SPLINE
SPL {X  -162.485, Y  +370.062, Z    +0.000, E1   +10.606, E3 +533690.258}
SPL {X  -162.818, Y  +379.636, Z    +0.000, E1    +5.115, E3 +533679.607}
SPL {X  -162.820, Y  +386.976, Z    +0.000, E1    +0.144, E3 +533678.706}
SPL {X  -162.820, Y  +391.982, Z    +0.000, E1    -3.443, E3 +533685.471}
SPL {X  -162.820, Y  +399.630, Z    +0.000, E1    -9.426, E3 +533687.978}
SPL {X  -162.820, Y  +408.127, Z    +0.000, E1   -18.417, E3 +533674.266}
SPL {X  -162.820, Y  +420.083, Z    +0.000, E1   -24.325, E3 +533694.742}
SPL {X  -162.820, Y  +428.527, Z    +0.000, E1   -26.988, E3 +533712.034}
SPL {X  -162.820, Y  +431.191, Z    +0.000, E1   -23.548, E3 +533746.887}
SPL {X  -162.820, Y  +432.946, Z    +0.000, E1   -22.795, E3 +533761.291}
SPL {X  -162.820, Y  +434.888, Z    +0.000, E1   -22.823, E3 +533770.697}
SPL {X  -162.820, Y  +436.834, Z    +0.000, E1   -22.779, E3 +533780.657}
SPL {X  -162.820, Y  +438.868, Z    +0.000, E1   -22.837, E3 +533790.311}
SPL {X  -162.820, Y  +441.351, Z    +0.000, E1   -22.805, E3 +533802.886}
SPL {X  -162.820, Y  +443.809, Z    +0.000, E1   -22.804, E3 +533815.052}
SPL {X  -162.820, Y  +446.105, Z    +0.000, E1   -22.815, E3 +533826.295}
SPL {X  -162.820, Y  +447.974, Z    +0.000, E1   -22.856, E3 +533835.198}
SPL {X  -162.820, Y  +449.911, Z    +0.000, E1   -22.774, E3 +533845.472}
SPL {X  -162.820, Y  +451.861, Z    +0.000, E1   -22.750, E3 +533855.320}
SPL {X  -162.820, Y  +454.167, Z    +0.000, E1   -22.842, E3 +533866.049}
SPL {X  -162.820, Y  +456.529, Z    +0.000, E1   -22.855, E3 +533877.578}
SPL {X  -162.820, Y  +458.725, Z    +0.000, E1   -22.793, E3 +533888.982}
SPL {X  -162.820, Y  +461.700, Z    +0.000, E1   -22.822, E3 +533903.605}
SPL {X  -162.820, Y  +464.633, Z    +0.000, E1   -22.813, E3 +533918.101}
SPL {X  -162.820, Y  +466.699, Z    +0.000, E1   -22.824, E3 +533928.147}
SPL {X  -162.820, Y  +468.655, Z    +0.000, E1   -22.858, E3 +533937.591}
SPL {X  -162.820, Y  +470.892, Z    +0.000, E1   -22.837, E3 +533948.830}
SPL {X  -162.820, Y  +472.726, Z    +0.000, E1   -22.777, E3 +533958.369}
SPL {X  -162.820, Y  +475.118, Z    +0.000, E1   -22.777, E3 +533970.340}
SPL {X  -162.820, Y  +478.177, Z    +0.000, E1   -22.834, E3 +533985.033}
SPL {X  -162.820, Y  +481.034, Z    +0.000, E1   -22.831, E3 +533999.170}
SPL {X  -162.820, Y  +483.391, Z    +0.000, E1   -22.793, E3 +534011.106}
SPL {X  -162.820, Y  +486.307, Z    +0.000, E1   -22.833, E3 +534025.360}
SPL {X  -162.820, Y  +488.828, Z    +0.000, E1   -22.793, E3 +534038.003}
SPL {X  -162.820, Y  +491.768, Z    +0.000, E1   -22.852, E3 +534052.300}
SPL {X  -162.820, Y  +495.526, Z    +0.000, E1   -22.833, E3 +534071.071}
SPL {X  -162.820, Y  +499.330, Z    +0.000, E1   -22.841, E3 +534089.852}
SPL {X  -162.820, Y  +503.049, Z    +0.000, E1   -22.823, E3 +534108.402}
SPL {X  -162.820, Y  +506.908, Z    +0.000, E1   -22.877, E3 +534127.072}
SPL {X  -162.820, Y  +510.068, Z    +0.000, E1   -22.761, E3 +534143.543}
SPL {X  -162.820, Y  +512.359, Z    +0.000, E1   -22.823, E3 +534154.275}
SPL {X  -162.820, Y  +513.873, Z    +0.000, E1   -22.800, E3 +534161.961}
SPL {X  -162.820, Y  +516.100, Z    +0.000, E1   -22.809, E3 +534173.038}
SPL {X  -162.820, Y  +518.662, Z    +0.000, E1   -22.847, E3 +534185.337}
SPL {X  -162.820, Y  +520.641, Z    +0.000, E1   -22.790, E3 +534195.578}
SPL {X  -162.820, Y  +523.535, Z    +0.000, E1   -22.857, E3 +534209.546}
SPL {X  -162.820, Y  +526.661, Z    +0.000, E1   -22.801, E3 +534225.371}
SPL {X  -162.820, Y  +528.725, Z    +0.000, E1   -22.770, E3 +534235.740}
SPL {X  -162.820, Y  +530.303, Z    +0.000, E1   -22.798, E3 +534243.359}
SPL {X  -162.820, Y  +532.614, Z    +0.000, E1   -22.828, E3 +534254.627}
SPL {X  -162.820, Y  +534.838, Z    +0.000, E1   -22.864, E3 +534265.256}
SPL {X  -162.820, Y  +536.882, Z    +0.000, E1   -22.782, E3 +534276.111}
SPL {X  -162.820, Y  +539.194, Z    +0.000, E1   -22.826, E3 +534287.160}
SPL {X  -162.820, Y  +541.555, Z    +0.000, E1   -22.817, E3 +534298.974}
SPL {X  -162.820, Y  +543.728, Z    +0.000, E1   -22.799, E3 +534309.832}
SPL {X  -162.820, Y  +545.925, Z    +0.000, E1   -22.803, E3 +534320.702}
SPL {X  -162.820, Y  +549.071, Z    +0.000, E1   -22.836, E3 +534336.229}
SPL {X  -162.820, Y  +553.089, Z    +0.000, E1   -22.838, E3 +534356.129}
SPL {X  -162.820, Y  +556.430, Z    +0.000, E1   -22.821, E3 +534372.630}
SPL {X  -162.820, Y  +558.974, Z    +0.000, E1   -22.806, E3 +534385.330}
SPL {X  -162.820, Y  +562.171, Z    +0.000, E1   -22.845, E3 +534401.028}
SPL {X  -162.820, Y  +565.170, Z    +0.000, E1   -22.801, E3 +534416.041}
SPL {X  -162.820, Y  +567.308, Z    +0.000, E1   -22.750, E3 +534427.057}
SPL {X  -162.820, Y  +570.378, Z    +0.000, E1   -22.843, E3 +534441.681}
SPL {X  -162.820, Y  +573.634, Z    +0.000, E1   -22.827, E3 +534457.825}
SPL {X  -162.820, Y  +576.228, Z    +0.000, E1   -22.814, E3 +534470.721}
SPL {X  -162.820, Y  +578.553, Z    +0.000, E1   -22.801, E3 +534482.337}
SPL {X  -162.820, Y  +581.064, Z    +0.000, E1   -22.823, E3 +534494.622}
SPL {X  -162.820, Y  +583.435, Z    +0.000, E1   -22.808, E3 +534506.443}
SPL {X  -162.820, Y  +585.410, Z    +0.000, E1   -22.764, E3 +534516.579}
SPL {X  -162.820, Y  +587.676, Z    +0.000, E1   -22.853, E3 +534527.094}
SPL {X  -162.820, Y  +590.707, Z    +0.000, E1   -22.855, E3 +534542.244}
SPL {X  -162.820, Y  +593.650, Z    +0.000, E1   -22.810, E3 +534557.004}
SPL {X  -162.820, Y  +595.830, Z    +0.000, E1   -22.828, E3 +534567.620}
SPL {X  -162.820, Y  +598.094, Z    +0.000, E1   -22.843, E3 +534578.733}
SPL {X  -162.820, Y  +600.420, Z    +0.000, E1   -22.826, E3 +534590.365}
SPL {X  -162.820, Y  +602.573, Z    +0.000, E1   -22.830, E3 +534600.950}
SPL {X  -162.820, Y  +604.828, Z    +0.000, E1   -22.784, E3 +534612.588}
SPL {X  -162.820, Y  +608.133, Z    +0.000, E1   -22.831, E3 +534628.706}
SPL {X  -162.820, Y  +611.103, Z    +0.000, E1   -22.785, E3 +534643.632}
SPL {X  -162.820, Y  +613.294, Z    +0.000, E1   -22.780, E3 +534654.505}
SPL {X  -162.820, Y  +615.356, Z    +0.000, E1   -22.799, E3 +534664.562}
SPL {X  -162.820, Y  +617.439, Z    +0.000, E1   -22.808, E3 +534674.820}
SPL {X  -162.820, Y  +619.665, Z    +0.000, E1   -22.817, E3 +534685.788}
SPL {X  -162.820, Y  +621.733, Z    +0.000, E1   -22.759, E3 +534696.512}
SPL {X  -162.820, Y  +624.076, Z    +0.000, E1   -22.774, E3 +534708.017}
SPL {X  -162.820, Y  +627.244, Z    +0.000, E1   -22.803, E3 +534723.700}
SPL {X  -162.820, Y  +630.349, Z    +0.000, E1   -22.766, E3 +534739.232}
SPL {X  -162.820, Y  +632.572, Z    +0.000, E1   -22.785, E3 +534750.038}
SPL {X  -162.820, Y  +634.507, Z    +0.000, E1   -22.784, E3 +534759.677}
SPL {X  -162.820, Y  +636.863, Z    +0.000, E1   -22.760, E3 +534771.599}
SPL {X  -162.820, Y  +640.111, Z    +0.000, E1   -22.809, E3 +534787.482}
SPL {X  -162.820, Y  +643.449, Z    +0.000, E1   -22.796, E3 +534804.000}
SPL {X  -162.820, Y  +645.630, Z    +0.000, E1   -22.795, E3 +534814.696}
SPL {X  -162.820, Y  +647.561, Z    +0.000, E1   -22.705, E3 +534825.147}
SPL {X  -162.820, Y  +651.051, Z    +0.000, E1   -22.833, E3 +534841.566}
SPL {X  -162.820, Y  +653.898, Z    +0.000, E1   -22.796, E3 +534855.752}
SPL {X  -162.820, Y  +656.161, Z    +0.000, E1   -22.812, E3 +534866.873}
SPL {X  -162.820, Y  +658.384, Z    +0.000, E1   -22.822, E3 +534877.740}
SPL {X  -162.820, Y  +660.215, Z    +0.000, E1   -22.649, E3 +534888.330}
SPL {X  -162.820, Y  +662.823, Z    +0.000, E1   -22.799, E3 +534900.038}
SPL {X  -162.820, Y  +665.862, Z    +0.000, E1   -22.864, E3 +534914.738}
SPL {X  -162.820, Y  +668.960, Z    +0.000, E1   -22.773, E3 +534930.688}
SPL {X  -162.820, Y  +672.333, Z    +0.000, E1   -22.837, E3 +534947.024}
SPL {X  -162.812, Y  +675.071, Z    +0.000, E1   -22.742, E3 +534961.170}
SPL {X  -162.773, Y  +677.428, Z    +0.000, E1   -22.762, E3 +534972.767}
SPL {X  -162.691, Y  +679.987, Z    +0.000, E1   -22.794, E3 +534985.180}
SPL {X  -162.604, Y  +681.880, Z    +0.000, E1   -22.691, E3 +534995.341}
SPL {X  -162.458, Y  +684.346, Z    +0.000, E1   -22.764, E3 +535007.135}
SPL {X  -162.296, Y  +686.547, Z    +0.000, E1   -22.660, E3 +535018.752}
SPL {X  -162.090, Y  +688.902, Z    +0.000, E1   -22.700, E3 +535030.260}
SPL {X  -161.474, Y  +694.390, Z    +0.000, E1   -24.298, E3 +535043.615}
SPL {X  -158.730, Y  +709.763, Z    +0.000, E1   -31.225, E3 +535054.954}
ENDSPLINE

SPLINE
SPL {X  -160.932, Y  +698.225, Z    +0.000, E1   -21.712, E3 +535086.063}
SPL {X  -161.917, Y  +690.622, Z    +0.000, E1   -16.445, E3 +535099.663}
ENDSPLINE

SPLINE
SPL {X  -161.349, Y  +695.340, Z    +0.000, E1   -18.625, E3 +535107.282}
ENDSPLINE

SPLINE
SPL {X  -162.534, Y  +683.153, Z    +0.000, E1   -10.475, E3 +535128.413}
SPL {X  -162.820, Y  +667.630, Z    +0.000, E1    -0.882, E3 +535122.389}
SPL {X  -162.820, Y  +661.883, Z    +0.000, E1    +3.373, E3 +535127.832}
SPL {X  -162.820, Y  +653.808, Z    +0.000, E1    +9.891, E3 +535125.524}
SPL {X  -162.820, Y  +632.548, Z    +0.000, E1   +27.446, E3 +535122.060}
ENDSPLINE

SPLINE
SPL {X  -162.820, Y  +638.080, Z    +0.000, E1   +18.858, E3 +535149.809}
ENDSPLINE

SPLINE
SPL {X  -162.820, Y  +623.278, Z    +0.000, E1   +28.723, E3 +535151.379}
SPL {X  -162.820, Y  +618.658, Z    +0.000, E1   +26.841, E3 +535179.988}
ENDSPLINE

SPLINE
SPL {X  -162.820, Y  +623.685, Z    +0.000, E1   +22.346, E3 +535192.295}
ENDSPLINE

SPLINE
SPL {X  -162.820, Y  +621.304, Z    +0.000, E1   +22.259, E3 +535205.110}
SPL {X  -162.820, Y  +618.758, Z    +0.000, E1   +22.239, E3 +535218.261}
SPL {X  -162.820, Y  +616.062, Z    +0.000, E1   +22.275, E3 +535231.681}
SPL {X  -162.820, Y  +613.536, Z    +0.000, E1   +22.242, E3 +535244.803}
SPL {X  -162.820, Y  +610.461, Z    +0.000, E1   +22.264, E3 +535260.434}
SPL {X  -162.820, Y  +607.796, Z    +0.000, E1   +22.261, E3 +535273.805}
SPL {X  -162.820, Y  +605.178, Z    +0.000, E1   +22.267, E3 +535287.289}
SPL {X  -162.820, Y  +602.350, Z    +0.000, E1   +22.224, E3 +535301.907}
SPL {X  -162.820, Y  +599.842, Z    +0.000, E1   +22.298, E3 +535314.058}
SPL {X  -162.820, Y  +597.194, Z    +0.000, E1   +22.253, E3 +535327.979}
SPL {X  -162.820, Y  +594.779, Z    +0.000, E1   +22.284, E3 +535339.883}
SPL {X  -162.820, Y  +592.389, Z    +0.000, E1   +22.245, E3 +535352.499}
SPL {X  -162.820, Y  +589.492, Z    +0.000, E1   +22.304, E3 +535366.684}
SPL {X  -162.820, Y  +587.447, Z    +0.000, E1   +22.279, E3 +535377.213}
SPL {X  -162.820, Y  +585.192, Z    +0.000, E1   +22.298, E3 +535388.623}
SPL {X  -162.820, Y  +582.610, Z    +0.000, E1   +22.234, E3 +535402.246}
SPL {X  -162.820, Y  +580.317, Z    +0.000, E1   +22.300, E3 +535413.300}
SPL {X  -162.820, Y  +578.878, Z    +0.000, E1   +22.272, E3 +535420.810}
SPL {X  -162.820, Y  +576.856, Z    +0.000, E1   +22.233, E3 +535431.568}
SPL {X  -162.820, Y  +574.811, Z    +0.000, E1   +22.236, E3 +535441.832}
SPL {X  -162.820, Y  +572.645, Z    +0.000, E1   +22.246, E3 +535452.927}
SPL {X  -162.820, Y  +570.282, Z    +0.000, E1   +22.231, E3 +535464.978}
SPL {X  -162.820, Y  +567.961, Z    +0.000, E1   +22.247, E3 +535476.767}
SPL {X  -162.820, Y  +564.506, Z    +0.000, E1   +22.298, E3 +535494.081}
SPL {X  -162.820, Y  +561.620, Z    +0.000, E1   +22.191, E3 +535509.462}
SPL {X  -162.820, Y  +559.515, Z    +0.000, E1   +22.273, E3 +535519.464}
SPL {X  -162.820, Y  +556.723, Z    +0.000, E1   +22.309, E3 +535533.548}
SPL {X  -162.820, Y  +554.378, Z    +0.000, E1   +22.288, E3 +535545.393}
SPL {X  -162.820, Y  +552.787, Z    +0.000, E1   +22.213, E3 +535554.215}
SPL {X  -162.820, Y  +550.871, Z    +0.000, E1   +22.229, E3 +535563.810}
SPL {X  -162.820, Y  +548.168, Z    +0.000, E1   +22.298, E3 +535577.146}
SPL {X  -162.820, Y  +545.860, Z    +0.000, E1   +22.216, E3 +535589.403}
SPL {X  -162.820, Y  +543.558, Z    +0.000, E1   +22.285, E3 +535600.634}
SPL {X  -162.820, Y  +541.633, Z    +0.000, E1   +22.257, E3 +535610.562}
SPL {X  -162.820, Y  +539.116, Z    +0.000, E1   +22.302, E3 +535623.172}
SPL {X  -162.820, Y  +535.523, Z    +0.000, E1   +22.266, E3 +535641.834}
SPL {X  -162.820, Y  +531.757, Z    +0.000, E1   +22.276, E3 +535660.889}
SPL {X  -162.820, Y  +527.980, Z    +0.000, E1   +22.326, E3 +535679.720}
SPL {X  -162.820, Y  +524.599, Z    +0.000, E1   +22.287, E3 +535697.117}
SPL {X  -162.820, Y  +522.011, Z    +0.000, E1   +22.282, E3 +535710.194}
SPL {X  -162.820, Y  +519.457, Z    +0.000, E1   +22.481, E3 +535721.483}
SPL {X  -162.820, Y  +506.285, Z    +0.000, E1   +28.538, E3 +535732.941}
SPL {X  -162.820, Y  +504.441, Z    +0.000, E1   +27.574, E3 +535747.284}
SPL {X  -162.820, Y  +502.813, Z    +0.000, E1   +26.013, E3 +535765.481}
SPL {X  -162.820, Y  +502.016, Z    +0.000, E1   +24.802, E3 +535777.824}
SPL {X  -162.820, Y  +501.060, Z    +0.000, E1   +24.081, E3 +535788.013}
SPL {X  -162.820, Y  +500.336, Z    +0.000, E1   +23.110, E3 +535799.153}
SPL {X  -162.820, Y  +499.240, Z    +0.000, E1   +22.316, E3 +535811.464}
SPL {X  -162.820, Y  +498.027, Z    +0.000, E1   +21.516, E3 +535824.372}
SPL {X  -162.820, Y  +495.897, Z    +0.000, E1   +21.662, E3 +535834.292}
SPL {X  -162.820, Y  +493.717, Z    +0.000, E1   +21.704, E3 +535845.398}
SPL {X  -162.820, Y  +491.396, Z    +0.000, E1   +21.707, E3 +535857.522}
SPL {X  -162.820, Y  +488.560, Z    +0.000, E1   +21.695, E3 +535872.632}
SPL {X  -162.820, Y  +485.661, Z    +0.000, E1   +21.712, E3 +535887.517}
SPL {X  -162.820, Y  +483.668, Z    +0.000, E1   +21.664, E3 +535898.344}
SPL {X  -162.820, Y  +481.739, Z    +0.000, E1   +21.704, E3 +535908.058}
SPL {X  -162.820, Y  +479.894, Z    +0.000, E1   +21.695, E3 +535917.845}
SPL {X  -162.820, Y  +477.685, Z    +0.000, E1   +21.656, E3 +535929.783}
SPL {X  -162.820, Y  +475.419, Z    +0.000, E1   +21.711, E3 +535941.136}
SPL {X  -162.820, Y  +473.301, Z    +0.000, E1   +21.712, E3 +535952.233}
SPL {X  -162.820, Y  +470.965, Z    +0.000, E1   +21.700, E3 +535964.578}
SPL {X  -162.820, Y  +469.036, Z    +0.000, E1   +21.695, E3 +535974.621}
SPL {X  -162.820, Y  +467.138, Z    +0.000, E1   +21.678, E3 +535984.793}
SPL {X  -162.820, Y  +465.011, Z    +0.000, E1   +21.692, E3 +535995.776}
SPL {X  -162.820, Y  +462.669, Z    +0.000, E1   +21.752, E3 +536007.556}
SPL {X  -162.820, Y  +460.725, Z    +0.000, E1   +21.689, E3 +536018.169}
SPL {X  -162.820, Y  +458.666, Z    +0.000, E1   +21.695, E3 +536028.981}
SPL {X  -162.820, Y  +456.431, Z    +0.000, E1   +21.708, E3 +536040.510}
SPL {X  -162.820, Y  +453.609, Z    +0.000, E1   +21.757, E3 +536055.044}
SPL {X  -162.820, Y  +450.610, Z    +0.000, E1   +21.698, E3 +536071.101}
SPL {X  -162.820, Y  +448.170, Z    +0.000, E1   +21.667, E3 +536084.122}
SPL {X  -162.820, Y  +446.246, Z    +0.000, E1   +21.696, E3 +536093.939}
SPL {X  -162.820, Y  +443.784, Z    +0.000, E1   +21.713, E3 +536106.726}
SPL {X  -162.820, Y  +440.567, Z    +0.000, E1   +21.731, E3 +536123.565}
SPL {X  -162.820, Y  +437.628, Z    +0.000, E1   +21.678, E3 +536139.229}
SPL {X  -162.820, Y  +434.473, Z    +0.000, E1   +21.747, E3 +536155.326}
SPL {X  -162.820, Y  +431.492, Z    +0.000, E1   +21.686, E3 +536171.274}
SPL {X  -162.820, Y  +429.074, Z    +0.000, E1   +21.710, E3 +536183.726}
SPL {X  -162.820, Y  +426.023, Z    +0.000, E1   +21.718, E3 +536199.794}
SPL {X  -162.820, Y  +422.986, Z    +0.000, E1   +21.685, E3 +536215.842}
SPL {X  -162.820, Y  +420.528, Z    +0.000, E1   +21.706, E3 +536228.492}
SPL {X  -162.820, Y  +418.116, Z    +0.000, E1   +21.761, E3 +536240.639}
SPL {X  -162.820, Y  +416.127, Z    +0.000, E1   +21.715, E3 +536251.344}
SPL {X  -162.820, Y  +414.361, Z    +0.000, E1   +21.613, E3 +536261.531}
SPL {X  -162.820, Y  +412.134, Z    +0.000, E1   +21.697, E3 +536272.476}
SPL {X  -162.820, Y  +409.248, Z    +0.000, E1   +21.741, E3 +536287.411}
SPL {X  -162.820, Y  +406.238, Z    +0.000, E1   +21.697, E3 +536303.379}
SPL {X  -162.820, Y  +404.001, Z    +0.000, E1   +21.723, E3 +536314.809}
SPL {X  -162.820, Y  +402.223, Z    +0.000, E1   +21.697, E3 +536324.294}
SPL {X  -162.820, Y  +400.348, Z    +0.000, E1   +21.713, E3 +536334.020}
SPL {X  -162.820, Y  +398.298, Z    +0.000, E1   +21.721, E3 +536344.635}
SPL {X  -162.820, Y  +396.371, Z    +0.000, E1   +21.713, E3 +536354.817}
SPL {X  -162.820, Y  +394.508, Z    +0.000, E1   +21.616, E3 +536365.373}
SPL {X  -162.820, Y  +392.435, Z    +0.000, E1   +21.681, E3 +536375.726}
SPL {X  -162.820, Y  +389.390, Z    +0.000, E1   +21.742, E3 +536391.333}
SPL {X  -162.820, Y  +386.818, Z    +0.000, E1   +21.679, E3 +536405.092}
SPL {X  -162.820, Y  +384.697, Z    +0.000, E1   +21.693, E3 +536416.162}
SPL {X  -162.820, Y  +382.288, Z    +0.000, E1   +21.742, E3 +536428.286}
SPL {X  -162.820, Y  +380.381, Z    +0.000, E1   +21.655, E3 +536439.010}
SPL {X  -162.808, Y  +378.512, Z    +0.000, E1   +21.736, E3 +536448.063}
SPL {X  -162.776, Y  +376.710, Z    +0.000, E1   +21.698, E3 +536457.862}
SPL {X  -162.707, Y  +374.438, Z    +0.000, E1   +21.688, E3 +536469.866}
SPL {X  -162.607, Y  +372.171, Z    +0.000, E1   +21.692, E3 +536481.666}
SPL {X  -162.494, Y  +370.197, Z    +0.000, E1   +21.655, E3 +536492.292}
SPL {X  -162.349, Y  +368.131, Z    +0.000, E1   +21.624, E3 +536503.410}
SPL {X  -162.161, Y  +365.866, Z    +0.000, E1   +21.642, E3 +536515.095}
SPL {X  -161.927, Y  +363.466, Z    +0.000, E1   +21.730, E3 +536526.867}
SPL {X  -160.290, Y  +351.907, Z    +0.000, E1   +27.562, E3 +536534.444}
SPL {X  -159.725, Y  +348.905, Z    +0.000, E1   +26.136, E3 +536559.679}
ENDSPLINE

SPLINE
SPL {X  -160.871, Y  +355.385, Z    +0.000, E1   +21.841, E3 +536568.522}
SPL {X  -161.833, Y  +362.603, Z    +0.000, E1   +17.021, E3 +536578.553}
ENDSPLINE

SPLINE
SPL {X  -160.786, Y  +354.842, Z    +0.000, E1   +19.274, E3 +536610.709}
ENDSPLINE

SPLINE
SPL {X  -162.485, Y  +370.062, Z    +0.000, E1   +10.606, E3 +536617.087}
SPL {X  -162.818, Y  +379.636, Z    +0.000, E1    +5.115, E3 +536606.436}
SPL {X  -162.820, Y  +386.976, Z    +0.000, E1    +0.144, E3 +536605.535}
SPL {X  -162.820, Y  +390.236, Z    +0.000, E1    -2.204, E3 +536611.594}
SPL {X  -162.820, Y  +393.415, Z    +0.000, E1    -4.587, E3 +536612.878}
SPL {X  -162.820, Y  +399.630, Z    +0.000, E1    -9.426, E3 +536614.807}
SPL {X  -162.820, Y  +408.127, Z    +0.000, E1   -18.417, E3 +536601.096}
SPL {X  -162.820, Y  +420.083, Z    +0.000, E1   -24.325, E3 +536621.571}
SPL {X  -162.820, Y  +428.527, Z    +0.000, E1   -26.988, E3 +536638.863}
SPL {X  -162.820, Y  +431.191, Z    +0.000, E1   -23.548, E3 +536673.716}
SPL {X  -162.820, Y  +432.946, Z    +0.000, E1   -22.795, E3 +536688.120}
SPL {X  -162.820, Y  +434.888, Z    +0.000, E1   -22.823, E3 +536697.527}
SPL {X  -162.820, Y  +436.834, Z    +0.000, E1   -22.779, E3 +536707.487}
SPL {X  -162.820, Y  +438.868, Z    +0.000, E1   -22.837, E3 +536717.140}
SPL {X  -162.820, Y  +441.351, Z    +0.000, E1   -22.805, E3 +536729.715}
SPL {X  -162.820, Y  +443.809, Z    +0.000, E1   -22.804, E3 +536741.882}
SPL {X  -162.820, Y  +446.105, Z    +0.000, E1   -22.815, E3 +536753.124}
SPL {X  -162.820, Y  +447.974, Z    +0.000, E1   -22.856, E3 +536762.027}
SPL {X  -162.820, Y  +449.911, Z    +0.000, E1   -22.774, E3 +536772.302}
SPL {X  -162.820, Y  +451.861, Z    +0.000, E1   -22.750, E3 +536782.149}
SPL {X  -162.820, Y  +454.167, Z    +0.000, E1   -22.842, E3 +536792.879}
SPL {X  -162.820, Y  +456.529, Z    +0.000, E1   -22.855, E3 +536804.407}
SPL {X  -162.820, Y  +458.725, Z    +0.000, E1   -22.793, E3 +536815.811}
SPL {X  -162.820, Y  +461.700, Z    +0.000, E1   -22.822, E3 +536830.434}
SPL {X  -162.820, Y  +464.633, Z    +0.000, E1   -22.813, E3 +536844.931}
SPL {X  -162.820, Y  +466.699, Z    +0.000, E1   -22.824, E3 +536854.977}
SPL {X  -162.820, Y  +468.655, Z    +0.000, E1   -22.858, E3 +536864.420}
SPL {X  -162.820, Y  +470.892, Z    +0.000, E1   -22.837, E3 +536875.659}
SPL {X  -162.820, Y  +473.485, Z    +0.000, E1   -22.806, E3 +536888.858}
SPL {X  -162.820, Y  +476.589, Z    +0.000, E1   -22.788, E3 +536904.379}
SPL {X  -162.820, Y  +478.914, Z    +0.000, E1   -22.821, E3 +536915.477}
SPL {X  -162.820, Y  +481.034, Z    +0.000, E1   -22.831, E3 +536926.000}
SPL {X  -162.820, Y  +484.256, Z    +0.000, E1   -22.840, E3 +536942.018}
SPL {X  -162.820, Y  +487.952, Z    +0.000, E1   -22.824, E3 +536960.448}
SPL {X  -162.820, Y  +491.768, Z    +0.000, E1   -22.852, E3 +536979.129}
SPL {X  -162.820, Y  +495.526, Z    +0.000, E1   -22.833, E3 +536997.900}
SPL {X  -162.820, Y  +499.330, Z    +0.000, E1   -22.841, E3 +537016.682}
SPL {X  -162.820, Y  +503.049, Z    +0.000, E1   -22.823, E3 +537035.231}
SPL {X  -162.820, Y  +506.908, Z    +0.000, E1   -22.877, E3 +537053.901}
SPL {X  -162.820, Y  +510.068, Z    +0.000, E1   -22.761, E3 +537070.373}
SPL {X  -162.820, Y  +512.359, Z    +0.000, E1   -22.823, E3 +537081.104}
SPL {X  -162.820, Y  +513.873, Z    +0.000, E1   -22.800, E3 +537088.791}
SPL {X  -162.820, Y  +516.100, Z    +0.000, E1   -22.809, E3 +537099.867}
SPL {X  -162.820, Y  +518.662, Z    +0.000, E1   -22.847, E3 +537112.166}
SPL {X  -162.820, Y  +520.641, Z    +0.000, E1   -22.790, E3 +537122.407}
SPL {X  -162.820, Y  +523.535, Z    +0.000, E1   -22.857, E3 +537136.376}
SPL {X  -162.820, Y  +526.661, Z    +0.000, E1   -22.801, E3 +537152.200}
SPL {X  -162.820, Y  +528.725, Z    +0.000, E1   -22.770, E3 +537162.569}
SPL {X  -162.820, Y  +530.303, Z    +0.000, E1   -22.798, E3 +537170.188}
SPL {X  -162.820, Y  +532.614, Z    +0.000, E1   -22.828, E3 +537181.457}
SPL {X  -162.820, Y  +534.838, Z    +0.000, E1   -22.864, E3 +537192.086}
SPL {X  -162.820, Y  +536.882, Z    +0.000, E1   -22.782, E3 +537202.941}
SPL {X  -162.820, Y  +539.194, Z    +0.000, E1   -22.826, E3 +537213.989}
SPL {X  -162.820, Y  +541.555, Z    +0.000, E1   -22.817, E3 +537225.803}
SPL {X  -162.820, Y  +543.728, Z    +0.000, E1   -22.799, E3 +537236.661}
SPL {X  -162.820, Y  +545.925, Z    +0.000, E1   -22.803, E3 +537247.531}
SPL {X  -162.820, Y  +548.328, Z    +0.000, E1   -22.796, E3 +537259.526}
SPL {X  -162.820, Y  +551.027, Z    +0.000, E1   -22.819, E3 +537272.719}
SPL {X  -162.820, Y  +553.721, Z    +0.000, E1   -22.807, E3 +537286.163}
SPL {X  -162.820, Y  +556.430, Z    +0.000, E1   -22.821, E3 +537299.459}
SPL {X  -162.820, Y  +559.675, Z    +0.000, E1   -22.837, E3 +537315.540}
SPL {X  -162.820, Y  +562.799, Z    +0.000, E1   -22.814, E3 +537331.046}
SPL {X  -162.820, Y  +565.170, Z    +0.000, E1   -22.801, E3 +537342.871}
SPL {X  -162.820, Y  +568.020, Z    +0.000, E1   -22.787, E3 +537357.257}
SPL {X  -162.820, Y  +570.992, Z    +0.000, E1   -22.834, E3 +537371.477}
SPL {X  -162.820, Y  +572.901, Z    +0.000, E1   -22.775, E3 +537381.345}
SPL {X  -162.820, Y  +575.638, Z    +0.000, E1   -22.855, E3 +537394.454}
SPL {X  -162.820, Y  +578.553, Z    +0.000, E1   -22.801, E3 +537409.167}
SPL {X  -162.820, Y  +581.064, Z    +0.000, E1   -22.823, E3 +537421.451}
SPL {X  -162.820, Y  +583.435, Z    +0.000, E1   -22.808, E3 +537433.273}
SPL {X  -162.820, Y  +585.410, Z    +0.000, E1   -22.764, E3 +537443.409}
SPL {X  -162.820, Y  +587.676, Z    +0.000, E1   -22.853, E3 +537453.923}
SPL {X  -162.820, Y  +589.682, Z    +0.000, E1   -22.776, E3 +537464.453}
SPL {X  -162.820, Y  +591.720, Z    +0.000, E1   -22.868, E3 +537473.764}
SPL {X  -162.820, Y  +593.650, Z    +0.000, E1   -22.810, E3 +537483.834}
SPL {X  -162.820, Y  +595.830, Z    +0.000, E1   -22.828, E3 +537494.449}
SPL {X  -162.820, Y  +598.094, Z    +0.000, E1   -22.843, E3 +537505.563}
SPL {X  -162.820, Y  +600.420, Z    +0.000, E1   -22.826, E3 +537517.194}
SPL {X  -162.820, Y  +602.573, Z    +0.000, E1   -22.830, E3 +537527.779}
SPL {X  -162.820, Y  +604.828, Z    +0.000, E1   -22.784, E3 +537539.417}
SPL {X  -162.820, Y  +607.142, Z    +0.000, E1   -22.808, E3 +537550.598}
SPL {X  -162.820, Y  +608.890, Z    +0.000, E1   -22.790, E3 +537559.423}
SPL {X  -162.820, Y  +611.103, Z    +0.000, E1   -22.785, E3 +537570.461}
SPL {X  -162.820, Y  +613.294, Z    +0.000, E1   -22.780, E3 +537581.334}
SPL {X  -162.820, Y  +615.356, Z    +0.000, E1   -22.799, E3 +537591.391}
SPL {X  -162.820, Y  +617.439, Z    +0.000, E1   -22.808, E3 +537601.649}
SPL {X  -162.820, Y  +619.665, Z    +0.000, E1   -22.817, E3 +537612.617}
SPL {X  -162.820, Y  +621.733, Z    +0.000, E1   -22.759, E3 +537623.342}
SPL {X  -162.820, Y  +624.076, Z    +0.000, E1   -22.774, E3 +537634.847}
SPL {X  -162.820, Y  +626.527, Z    +0.000, E1   -22.768, E3 +537647.089}
SPL {X  -162.820, Y  +629.758, Z    +0.000, E1   -22.800, E3 +537663.018}
SPL {X  -162.820, Y  +632.572, Z    +0.000, E1   -22.785, E3 +537676.867}
SPL {X  -162.820, Y  +634.507, Z    +0.000, E1   -22.784, E3 +537686.506}
SPL {X  -162.820, Y  +636.863, Z    +0.000, E1   -22.760, E3 +537698.429}
SPL {X  -162.820, Y  +639.254, Z    +0.000, E1   -22.767, E3 +537710.212}
SPL {X  -162.820, Y  +641.888, Z    +0.000, E1   -22.790, E3 +537723.159}
SPL {X  -162.820, Y  +644.915, Z    +0.000, E1   -22.818, E3 +537737.934}
SPL {X  -162.820, Y  +647.561, Z    +0.000, E1   -22.705, E3 +537751.976}
SPL {X  -162.820, Y  +649.758, Z    +0.000, E1   -22.780, E3 +537762.166}
SPL {X  -162.820, Y  +651.708, Z    +0.000, E1   -22.810, E3 +537771.660}
SPL {X  -162.820, Y  +653.898, Z    +0.000, E1   -22.796, E3 +537782.581}
SPL {X  -162.820, Y  +656.161, Z    +0.000, E1   -22.812, E3 +537793.703}
SPL {X  -162.820, Y  +658.384, Z    +0.000, E1   -22.822, E3 +537804.569}
SPL {X  -162.820, Y  +660.215, Z    +0.000, E1   -22.649, E3 +537815.159}
SPL {X  -162.820, Y  +662.823, Z    +0.000, E1   -22.799, E3 +537826.867}
SPL {X  -162.820, Y  +665.862, Z    +0.000, E1   -22.864, E3 +537841.567}
SPL {X  -162.820, Y  +668.960, Z    +0.000, E1   -22.773, E3 +537857.518}
SPL {X  -162.820, Y  +672.333, Z    +0.000, E1   -22.837, E3 +537873.854}
SPL {X  -162.812, Y  +675.071, Z    +0.000, E1   -22.742, E3 +537887.999}
SPL {X  -162.773, Y  +677.428, Z    +0.000, E1   -22.762, E3 +537899.596}
SPL {X  -162.691, Y  +679.987, Z    +0.000, E1   -22.794, E3 +537912.010}
SPL {X  -162.604, Y  +681.880, Z    +0.000, E1   -22.691, E3 +537922.170}
SPL {X  -162.458, Y  +684.346, Z    +0.000, E1   -22.764, E3 +537933.964}
SPL {X  -162.296, Y  +686.547, Z    +0.000, E1   -22.660, E3 +537945.581}
SPL {X  -162.090, Y  +688.902, Z    +0.000, E1   -22.700, E3 +537957.089}
SPL {X  -161.474, Y  +694.390, Z    +0.000, E1   -24.298, E3 +537970.444}
SPL {X  -158.553, Y  +710.529, Z    +0.000, E1   -30.890, E3 +537987.006}
ENDSPLINE

SPLINE
SPL {X  -161.215, Y  +696.305, Z    +0.000, E1   -20.575, E3 +538013.587}
SPL {X  -161.691, Y  +692.643, Z    +0.000, E1   -17.369, E3 +538029.775}
SPL {X  -162.534, Y  +683.153, Z    +0.000, E1   -10.475, E3 +538055.242}
SPL {X  -162.820, Y  +667.630, Z    +0.000, E1    -0.882, E3 +538049.218}
SPL {X  -162.820, Y  +661.883, Z    +0.000, E1    +3.373, E3 +538054.662}
SPL {X  -162.820, Y  +653.808, Z    +0.000, E1    +9.891, E3 +538052.353}
SPL {X  -162.820, Y  +632.548, Z    +0.000, E1   +27.446, E3 +538048.890}
ENDSPLINE

SPLINE
SPL {X  -162.820, Y  +638.080, Z    +0.000, E1   +18.858, E3 +538076.638}
ENDSPLINE

SPLINE
SPL {X  -162.820, Y  +623.278, Z    +0.000, E1   +28.723, E3 +538078.209}
SPL {X  -162.820, Y  +618.658, Z    +0.000, E1   +26.841, E3 +538106.817}
ENDSPLINE

SPLINE
SPL {X  -162.820, Y  +623.685, Z    +0.000, E1   +22.346, E3 +538119.124}
ENDSPLINE

SPLINE
SPL {X  -162.820, Y  +621.304, Z    +0.000, E1   +22.259, E3 +538131.939}
SPL {X  -162.820, Y  +618.758, Z    +0.000, E1   +22.239, E3 +538145.090}
SPL {X  -162.820, Y  +616.062, Z    +0.000, E1   +22.275, E3 +538158.511}
SPL {X  -162.820, Y  +613.536, Z    +0.000, E1   +22.242, E3 +538171.632}
SPL {X  -162.820, Y  +611.128, Z    +0.000, E1   +22.252, E3 +538183.803}
SPL {X  -162.820, Y  +608.428, Z    +0.000, E1   +22.255, E3 +538197.586}
SPL {X  -162.820, Y  +605.984, Z    +0.000, E1   +22.221, E3 +538210.223}
SPL {X  -162.820, Y  +603.020, Z    +0.000, E1   +22.272, E3 +538225.122}
SPL {X  -162.820, Y  +599.168, Z    +0.000, E1   +22.310, E3 +538244.390}
SPL {X  -162.820, Y  +596.569, Z    +0.000, E1   +22.222, E3 +538258.112}
SPL {X  -162.820, Y  +594.115, Z    +0.000, E1   +22.273, E3 +538270.337}
SPL {X  -162.820, Y  +591.721, Z    +0.000, E1   +22.239, E3 +538282.652}
SPL {X  -162.820, Y  +589.492, Z    +0.000, E1   +22.304, E3 +538293.513}
SPL {X  -162.820, Y  +587.447, Z    +0.000, E1   +22.279, E3 +538304.042}
SPL {X  -162.820, Y  +585.192, Z    +0.000, E1   +22.298, E3 +538315.452}
SPL {X  -162.820, Y  +582.610, Z    +0.000, E1   +22.234, E3 +538329.076}
SPL {X  -162.820, Y  +580.317, Z    +0.000, E1   +22.300, E3 +538340.130}
SPL {X  -162.820, Y  +578.878, Z    +0.000, E1   +22.272, E3 +538347.639}
SPL {X  -162.820, Y  +576.856, Z    +0.000, E1   +22.233, E3 +538358.397}
SPL {X  -162.820, Y  +573.830, Z    +0.000, E1   +22.272, E3 +538373.533}
SPL {X  -162.820, Y  +570.852, Z    +0.000, E1   +22.234, E3 +538388.993}
SPL {X  -162.820, Y  +568.608, Z    +0.000, E1   +22.253, E3 +538400.126}
SPL {X  -162.820, Y  +565.838, Z    +0.000, E1   +22.271, E3 +538414.357}
SPL {X  -162.820, Y  +562.162, Z    +0.000, E1   +22.252, E3 +538433.175}
SPL {X  -162.820, Y  +558.919, Z    +0.000, E1   +22.286, E3 +538449.338}
SPL {X  -162.820, Y  +555.548, Z    +0.000, E1   +22.322, E3 +538466.247}
SPL {X  -162.820, Y  +552.787, Z    +0.000, E1   +22.213, E3 +538481.044}
SPL {X  -162.820, Y  +550.136, Z    +0.000, E1   +22.258, E3 +538494.278}
SPL {X  -162.820, Y  +546.694, Z    +0.000, E1   +22.290, E3 +538511.600}
SPL {X  -162.820, Y  +543.558, Z    +0.000, E1   +22.285, E3 +538527.463}
SPL {X  -162.820, Y  +541.633, Z    +0.000, E1   +22.257, E3 +538537.391}
SPL {X  -162.820, Y  +539.116, Z    +0.000, E1   +22.302, E3 +538550.002}
SPL {X  -162.820, Y  +536.913, Z    +0.000, E1   +22.192, E3 +538561.926}
SPL {X  -162.820, Y  +534.880, Z    +0.000, E1   +22.252, E3 +538571.880}
SPL {X  -162.820, Y  +532.896, Z    +0.000, E1   +22.234, E3 +538582.040}
SPL {X  -162.820, Y  +531.056, Z    +0.000, E1   +22.251, E3 +538591.322}
SPL {X  -162.820, Y  +528.708, Z    +0.000, E1   +22.319, E3 +538602.704}
SPL {X  -162.820, Y  +525.932, Z    +0.000, E1   +22.258, E3 +538617.460}
SPL {X  -162.820, Y  +522.524, Z    +0.000, E1   +22.326, E3 +538634.184}
SPL {X  -162.820, Y  +519.457, Z    +0.000, E1   +22.481, E3 +538648.313}
SPL {X  -162.820, Y  +506.285, Z    +0.000, E1   +28.538, E3 +538659.771}
SPL {X  -162.820, Y  +504.441, Z    +0.000, E1   +27.574, E3 +538674.113}
SPL {X  -162.820, Y  +502.813, Z    +0.000, E1   +26.013, E3 +538692.310}
SPL {X  -162.820, Y  +502.016, Z    +0.000, E1   +24.802, E3 +538704.653}
SPL {X  -162.820, Y  +501.060, Z    +0.000, E1   +24.081, E3 +538714.843}
SPL {X  -162.820, Y  +499.934, Z    +0.000, E1   +22.814, E3 +538730.711}
SPL {X  -162.820, Y  +498.303, Z    +0.000, E1   +21.749, E3 +538747.967}
SPL {X  -162.820, Y  +495.897, Z    +0.000, E1   +21.662, E3 +538761.121}
SPL {X  -162.820, Y  +493.717, Z    +0.000, E1   +21.704, E3 +538772.227}
SPL {X  -162.820, Y  +491.396, Z    +0.000, E1   +21.707, E3 +538784.351}
SPL {X  -162.820, Y  +489.485, Z    +0.000, E1   +21.661, E3 +538794.699}
SPL {X  -162.820, Y  +487.723, Z    +0.000, E1   +21.665, E3 +538803.903}
SPL {X  -162.820, Y  +485.661, Z    +0.000, E1   +21.712, E3 +538814.346}
SPL {X  -162.820, Y  +482.775, Z    +0.000, E1   +21.716, E3 +538829.598}
SPL {X  -162.820, Y  +479.894, Z    +0.000, E1   +21.695, E3 +538844.675}
SPL {X  -162.820, Y  +477.685, Z    +0.000, E1   +21.656, E3 +538856.612}
SPL {X  -162.820, Y  +475.419, Z    +0.000, E1   +21.711, E3 +538867.965}
SPL {X  -162.820, Y  +473.301, Z    +0.000, E1   +21.712, E3 +538879.062}
SPL {X  -162.820, Y  +470.965, Z    +0.000, E1   +21.700, E3 +538891.407}
SPL {X  -162.820, Y  +469.036, Z    +0.000, E1   +21.695, E3 +538901.451}
SPL {X  -162.820, Y  +467.138, Z    +0.000, E1   +21.678, E3 +538911.622}
SPL {X  -162.820, Y  +465.011, Z    +0.000, E1   +21.692, E3 +538922.605}
SPL {X  -162.820, Y  +462.669, Z    +0.000, E1   +21.752, E3 +538934.385}
SPL {X  -162.820, Y  +460.725, Z    +0.000, E1   +21.689, E3 +538944.998}
SPL {X  -162.820, Y  +458.666, Z    +0.000, E1   +21.695, E3 +538955.810}
SPL {X  -162.820, Y  +456.431, Z    +0.000, E1   +21.708, E3 +538967.339}
SPL {X  -162.820, Y  +454.628, Z    +0.000, E1   +21.674, E3 +538977.057}
SPL {X  -162.820, Y  +452.690, Z    +0.000, E1   +21.773, E3 +538986.331}
SPL {X  -162.820, Y  +450.610, Z    +0.000, E1   +21.698, E3 +538997.930}
SPL {X  -162.820, Y  +448.170, Z    +0.000, E1   +21.667, E3 +539010.951}
SPL {X  -162.820, Y  +445.508, Z    +0.000, E1   +21.732, E3 +539024.469}
SPL {X  -162.820, Y  +442.443, Z    +0.000, E1   +21.712, E3 +539040.590}
SPL {X  -162.820, Y  +439.933, Z    +0.000, E1   +21.690, E3 +539053.871}
SPL {X  -162.820, Y  +437.628, Z    +0.000, E1   +21.678, E3 +539066.059}
SPL {X  -162.820, Y  +434.473, Z    +0.000, E1   +21.747, E3 +539082.155}
SPL {X  -162.820, Y  +431.492, Z    +0.000, E1   +21.686, E3 +539098.104}
SPL {X  -162.820, Y  +429.074, Z    +0.000, E1   +21.710, E3 +539110.556}
SPL {X  -162.820, Y  +426.023, Z    +0.000, E1   +21.718, E3 +539126.623}
SPL {X  -162.820, Y  +422.986, Z    +0.000, E1   +21.685, E3 +539142.671}
SPL {X  -162.820, Y  +420.528, Z    +0.000, E1   +21.706, E3 +539155.321}
SPL {X  -162.820, Y  +418.116, Z    +0.000, E1   +21.761, E3 +539167.468}
SPL {X  -162.820, Y  +416.127, Z    +0.000, E1   +21.715, E3 +539178.173}
SPL {X  -162.820, Y  +414.361, Z    +0.000, E1   +21.613, E3 +539188.360}
SPL {X  -162.820, Y  +411.450, Z    +0.000, E1   +21.710, E3 +539202.934}
SPL {X  -162.820, Y  +408.590, Z    +0.000, E1   +21.735, E3 +539217.559}
SPL {X  -162.820, Y  +406.238, Z    +0.000, E1   +21.697, E3 +539230.208}
SPL {X  -162.820, Y  +403.166, Z    +0.000, E1   +21.746, E3 +539246.014}
SPL {X  -162.820, Y  +400.348, Z    +0.000, E1   +21.713, E3 +539260.849}
SPL {X  -162.820, Y  +398.298, Z    +0.000, E1   +21.721, E3 +539271.465}
SPL {X  -162.820, Y  +396.371, Z    +0.000, E1   +21.713, E3 +539281.647}
SPL {X  -162.820, Y  +394.508, Z    +0.000, E1   +21.616, E3 +539292.202}
SPL {X  -162.820, Y  +391.777, Z    +0.000, E1   +21.714, E3 +539305.861}
SPL {X  -162.820, Y  +388.822, Z    +0.000, E1   +21.717, E3 +539321.181}
SPL {X  -162.820, Y  +386.818, Z    +0.000, E1   +21.679, E3 +539331.921}
SPL {X  -162.820, Y  +384.697, Z    +0.000, E1   +21.693, E3 +539342.991}
SPL {X  -162.820, Y  +382.288, Z    +0.000, E1   +21.742, E3 +539355.115}
SPL {X  -162.817, Y  +379.520, Z    +0.000, E1   +21.723, E3 +539369.952}
SPL {X  -162.776, Y  +376.710, Z    +0.000, E1   +21.698, E3 +539384.691}
SPL {X  -162.707, Y  +374.438, Z    +0.000, E1   +21.688, E3 +539396.695}
SPL {X  -162.607, Y  +372.171, Z    +0.000, E1   +21.692, E3 +539408.495}
SPL {X  -162.494, Y  +370.197, Z    +0.000, E1   +21.655, E3 +539419.121}
SPL {X  -162.349, Y  +368.131, Z    +0.000, E1   +21.624, E3 +539430.239}
SPL {X  -162.161, Y  +365.866, Z    +0.000, E1   +21.642, E3 +539441.924}
SPL {X  -161.651, Y  +361.024, Z    +0.000, E1   +22.970, E3 +539455.348}
SPL {X  -160.281, Y  +351.857, Z    +0.000, E1   +24.243, E3 +539490.687}
ENDSPLINE

SPLINE
SPL {X  -161.833, Y  +362.603, Z    +0.000, E1   +17.021, E3 +539505.383}
ENDSPLINE

SPLINE
SPL {X  -160.786, Y  +354.842, Z    +0.000, E1   +19.274, E3 +539537.538}
ENDSPLINE

SPLINE
SPL {X  -162.485, Y  +370.062, Z    +0.000, E1   +10.606, E3 +539543.916}
SPL {X  -162.818, Y  +379.636, Z    +0.000, E1    +5.115, E3 +539533.265}
SPL {X  -162.820, Y  +386.976, Z    +0.000, E1    +0.144, E3 +539532.364}
SPL {X  -162.820, Y  +390.236, Z    +0.000, E1    -2.204, E3 +539538.423}
SPL {X  -162.820, Y  +393.415, Z    +0.000, E1    -4.587, E3 +539539.707}
SPL {X  -162.820, Y  +399.630, Z    +0.000, E1    -9.426, E3 +539541.637}
SPL {X  -162.820, Y  +408.127, Z    +0.000, E1   -18.417, E3 +539527.925}
SPL {X  -162.820, Y  +420.083, Z    +0.000, E1   -24.325, E3 +539548.400}
SPL {X  -162.820, Y  +428.527, Z    +0.000, E1   -26.988, E3 +539565.693}
SPL {X  -162.820, Y  +431.336, Z    +0.000, E1   -24.162, E3 +539595.903}
SPL {X  -162.820, Y  +432.048, Z    +0.000, E1   -22.832, E3 +539610.406}
SPL {X  -162.820, Y  +434.888, Z    +0.000, E1   -22.823, E3 +539624.356}
SPL {X  -162.820, Y  +436.834, Z    +0.000, E1   -22.779, E3 +539634.316}
SPL {X  -162.820, Y  +438.868, Z    +0.000, E1   -22.837, E3 +539643.969}
SPL {X  -162.820, Y  +441.351, Z    +0.000, E1   -22.805, E3 +539656.545}
SPL {X  -162.820, Y  +443.809, Z    +0.000, E1   -22.804, E3 +539668.711}
SPL {X  -162.820, Y  +446.105, Z    +0.000, E1   -22.815, E3 +539679.953}
SPL {X  -162.820, Y  +447.974, Z    +0.000, E1   -22.856, E3 +539688.856}
SPL {X  -162.820, Y  +449.911, Z    +0.000, E1   -22.774, E3 +539699.131}
SPL {X  -162.820, Y  +451.861, Z    +0.000, E1   -22.750, E3 +539708.978}
SPL {X  -162.820, Y  +454.167, Z    +0.000, E1   -22.842, E3 +539719.708}
SPL {X  -162.820, Y  +456.529, Z    +0.000, E1   -22.855, E3 +539731.236}
SPL {X  -162.820, Y  +458.725, Z    +0.000, E1   -22.793, E3 +539742.641}
SPL {X  -162.820, Y  +461.700, Z    +0.000, E1   -22.822, E3 +539757.263}
SPL {X  -162.820, Y  +464.633, Z    +0.000, E1   -22.813, E3 +539771.760}
SPL {X  -162.820, Y  +466.699, Z    +0.000, E1   -22.824, E3 +539781.806}
SPL {X  -162.820, Y  +468.655, Z    +0.000, E1   -22.858, E3 +539791.250}
SPL {X  -162.820, Y  +470.892, Z    +0.000, E1   -22.837, E3 +539802.488}
SPL {X  -162.820, Y  +473.485, Z    +0.000, E1   -22.806, E3 +539815.687}
SPL {X  -162.820, Y  +476.589, Z    +0.000, E1   -22.788, E3 +539831.209}
SPL {X  -162.820, Y  +478.914, Z    +0.000, E1   -22.821, E3 +539842.307}
SPL {X  -162.820, Y  +481.034, Z    +0.000, E1   -22.831, E3 +539852.829}
SPL {X  -162.820, Y  +484.256, Z    +0.000, E1   -22.840, E3 +539868.848}
SPL {X  -162.820, Y  +487.014, Z    +0.000, E1   -22.789, E3 +539882.715}
SPL {X  -162.820, Y  +489.750, Z    +0.000, E1   -22.832, E3 +539896.089}
SPL {X  -162.820, Y  +493.233, Z    +0.000, E1   -22.844, E3 +539913.226}
SPL {X  -162.820, Y  +496.150, Z    +0.000, E1   -22.796, E3 +539927.945}
SPL {X  -162.820, Y  +498.661, Z    +0.000, E1   -22.828, E3 +539940.126}
SPL {X  -162.820, Y  +501.761, Z    +0.000, E1   -22.820, E3 +539955.695}
SPL {X  -162.820, Y  +505.323, Z    +0.000, E1   -22.838, E3 +539973.142}
SPL {X  -162.820, Y  +507.875, Z    +0.000, E1   -22.849, E3 +539985.509}
SPL {X  -162.820, Y  +510.068, Z    +0.000, E1   -22.761, E3 +539997.202}
SPL {X  -162.820, Y  +512.359, Z    +0.000, E1   -22.823, E3 +540007.933}
SPL {X  -162.820, Y  +514.562, Z    +0.000, E1   -22.806, E3 +540019.120}
SPL {X  -162.820, Y  +517.952, Z    +0.000, E1   -22.864, E3 +540035.518}
SPL {X  -162.820, Y  +520.641, Z    +0.000, E1   -22.790, E3 +540049.236}
SPL {X  -162.820, Y  +522.740, Z    +0.000, E1   -22.811, E3 +540059.479}
SPL {X  -162.820, Y  +524.628, Z    +0.000, E1   -22.846, E3 +540068.474}
SPL {X  -162.820, Y  +526.661, Z    +0.000, E1   -22.801, E3 +540079.029}
SPL {X  -162.820, Y  +529.662, Z    +0.000, E1   -22.810, E3 +540093.880}
SPL {X  -162.820, Y  +532.614, Z    +0.000, E1   -22.828, E3 +540108.286}
SPL {X  -162.820, Y  +534.838, Z    +0.000, E1   -22.864, E3 +540118.915}
SPL {X  -162.820, Y  +536.882, Z    +0.000, E1   -22.782, E3 +540129.770}
SPL {X  -162.820, Y  +539.194, Z    +0.000, E1   -22.826, E3 +540140.818}
SPL {X  -162.820, Y  +541.555, Z    +0.000, E1   -22.817, E3 +540152.633}
SPL {X  -162.820, Y  +543.728, Z    +0.000, E1   -22.799, E3 +540163.490}
SPL {X  -162.820, Y  +545.925, Z    +0.000, E1   -22.803, E3 +540174.360}
SPL {X  -162.820, Y  +548.328, Z    +0.000, E1   -22.796, E3 +540186.356}
SPL {X  -162.820, Y  +551.027, Z    +0.000, E1   -22.819, E3 +540199.549}
SPL {X  -162.820, Y  +553.721, Z    +0.000, E1   -22.807, E3 +540212.993}
SPL {X  -162.820, Y  +556.430, Z    +0.000, E1   -22.821, E3 +540226.289}
SPL {X  -162.820, Y  +559.675, Z    +0.000, E1   -22.837, E3 +540242.369}
SPL {X  -162.820, Y  +562.799, Z    +0.000, E1   -22.814, E3 +540257.875}
SPL {X  -162.820, Y  +565.170, Z    +0.000, E1   -22.801, E3 +540269.700}
SPL {X  -162.820, Y  +568.020, Z    +0.000, E1   -22.787, E3 +540284.087}
SPL {X  -162.820, Y  +570.992, Z    +0.000, E1   -22.834, E3 +540298.306}
SPL {X  -162.820, Y  +572.901, Z    +0.000, E1   -22.775, E3 +540308.174}
SPL {X  -162.820, Y  +575.638, Z    +0.000, E1   -22.855, E3 +540321.284}
SPL {X  -162.820, Y  +578.553, Z    +0.000, E1   -22.801, E3 +540335.996}
SPL {X  -162.820, Y  +581.064, Z    +0.000, E1   -22.823, E3 +540348.280}
SPL {X  -162.820, Y  +583.435, Z    +0.000, E1   -22.808, E3 +540360.102}
SPL {X  -162.820, Y  +585.410, Z    +0.000, E1   -22.764, E3 +540370.238}
SPL {X  -162.820, Y  +587.676, Z    +0.000, E1   -22.853, E3 +540380.752}
SPL {X  -162.820, Y  +589.682, Z    +0.000, E1   -22.776, E3 +540391.282}
SPL {X  -162.820, Y  +591.720, Z    +0.000, E1   -22.868, E3 +540400.593}
SPL {X  -162.820, Y  +593.650, Z    +0.000, E1   -22.810, E3 +540410.663}
SPL {X  -162.820, Y  +595.830, Z    +0.000, E1   -22.828, E3 +540421.279}
SPL {X  -162.820, Y  +598.094, Z    +0.000, E1   -22.843, E3 +540432.392}
SPL {X  -162.820, Y  +600.420, Z    +0.000, E1   -22.826, E3 +540444.023}
SPL {X  -162.820, Y  +602.573, Z    +0.000, E1   -22.830, E3 +540454.608}
SPL {X  -162.820, Y  +604.828, Z    +0.000, E1   -22.784, E3 +540466.247}
SPL {X  -162.820, Y  +607.142, Z    +0.000, E1   -22.808, E3 +540477.428}
SPL {X  -162.820, Y  +608.890, Z    +0.000, E1   -22.790, E3 +540486.252}
SPL {X  -162.820, Y  +611.103, Z    +0.000, E1   -22.785, E3 +540497.290}
SPL {X  -162.820, Y  +613.294, Z    +0.000, E1   -22.780, E3 +540508.163}
SPL {X  -162.820, Y  +615.356, Z    +0.000, E1   -22.799, E3 +540518.221}
SPL {X  -162.820, Y  +617.439, Z    +0.000, E1   -22.808, E3 +540528.479}
SPL {X  -162.820, Y  +619.665, Z    +0.000, E1   -22.817, E3 +540539.447}
SPL {X  -162.820, Y  +621.733, Z    +0.000, E1   -22.759, E3 +540550.171}
SPL {X  -162.820, Y  +624.076, Z    +0.000, E1   -22.774, E3 +540561.676}
SPL {X  -162.820, Y  +627.244, Z    +0.000, E1   -22.803, E3 +540577.358}
SPL {X  -162.820, Y  +630.349, Z    +0.000, E1   -22.766, E3 +540592.890}
SPL {X  -162.820, Y  +632.572, Z    +0.000, E1   -22.785, E3 +540603.697}
SPL {X  -162.820, Y  +634.507, Z    +0.000, E1   -22.784, E3 +540613.336}
SPL {X  -162.820, Y  +636.863, Z    +0.000, E1   -22.760, E3 +540625.258}
SPL {X  -162.820, Y  +640.111, Z    +0.000, E1   -22.809, E3 +540641.141}
SPL {X  -162.820, Y  +643.449, Z    +0.000, E1   -22.796, E3 +540657.658}
SPL {X  -162.820, Y  +645.630, Z    +0.000, E1   -22.795, E3 +540668.354}
SPL {X  -162.820, Y  +647.561, Z    +0.000, E1   -22.705, E3 +540678.805}
SPL {X  -162.820, Y  +649.758, Z    +0.000, E1   -22.780, E3 +540688.995}
SPL {X  -162.820, Y  +651.708, Z    +0.000, E1   -22.810, E3 +540698.490}
SPL {X  -162.820, Y  +653.898, Z    +0.000, E1   -22.796, E3 +540709.410}
SPL {X  -162.820, Y  +656.161, Z    +0.000, E1   -22.812, E3 +540720.532}
SPL {X  -162.820, Y  +658.384, Z    +0.000, E1   -22.822, E3 +540731.398}
SPL {X  -162.820, Y  +660.215, Z    +0.000, E1   -22.649, E3 +540741.989}
SPL {X  -162.820, Y  +662.823, Z    +0.000, E1   -22.799, E3 +540753.697}
SPL {X  -162.820, Y  +665.862, Z    +0.000, E1   -22.864, E3 +540768.396}
SPL {X  -162.820, Y  +668.960, Z    +0.000, E1   -22.773, E3 +540784.347}
SPL {X  -162.820, Y  +671.605, Z    +0.000, E1   -22.777, E3 +540797.421}
SPL {X  -162.817, Y  +674.515, Z    +0.000, E1   -22.816, E3 +540811.618}
SPL {X  -162.773, Y  +677.428, Z    +0.000, E1   -22.762, E3 +540826.426}
SPL {X  -162.691, Y  +679.987, Z    +0.000, E1   -22.794, E3 +540838.839}
SPL {X  -162.604, Y  +681.880, Z    +0.000, E1   -22.691, E3 +540849.000}
SPL {X  -162.458, Y  +684.346, Z    +0.000, E1   -22.764, E3 +540860.793}
SPL {X  -162.296, Y  +686.547, Z    +0.000, E1   -22.660, E3 +540872.410}
SPL {X  -162.090, Y  +688.902, Z    +0.000, E1   -22.700, E3 +540883.918}
SPL {X  -161.474, Y  +694.390, Z    +0.000, E1   -24.298, E3 +540897.273}
SPL {X  -158.553, Y  +710.529, Z    +0.000, E1   -30.890, E3 +540913.835}
ENDSPLINE

SPLINE
SPL {X  -161.215, Y  +696.305, Z    +0.000, E1   -20.575, E3 +540940.416}
SPL {X  -161.691, Y  +692.643, Z    +0.000, E1   -17.369, E3 +540956.604}
SPL {X  -162.534, Y  +683.153, Z    +0.000, E1   -10.475, E3 +540982.071}
SPL {X  -162.820, Y  +667.630, Z    +0.000, E1    -0.882, E3 +540976.048}
SPL {X  -162.820, Y  +661.883, Z    +0.000, E1    +3.373, E3 +540981.491}
SPL {X  -162.820, Y  +653.808, Z    +0.000, E1    +9.891, E3 +540979.182}
SPL {X  -162.820, Y  +632.548, Z    +0.000, E1   +27.446, E3 +540975.719}
ENDSPLINE

SPLINE
SPL {X  -162.820, Y  +638.080, Z    +0.000, E1   +18.858, E3 +541003.467}
ENDSPLINE

SPLINE
SPL {X  -162.820, Y  +623.278, Z    +0.000, E1   +28.723, E3 +541005.038}
SPL {X  -162.820, Y  +618.658, Z    +0.000, E1   +26.841, E3 +541033.647}
ENDSPLINE

SPLINE
SPL {X  -162.820, Y  +623.685, Z    +0.000, E1   +22.346, E3 +541045.954}
ENDSPLINE

SPLINE
SPL {X  -162.820, Y  +621.304, Z    +0.000, E1   +22.259, E3 +541058.769}
SPL {X  -162.820, Y  +618.758, Z    +0.000, E1   +22.239, E3 +541071.919}
SPL {X  -162.820, Y  +616.062, Z    +0.000, E1   +22.275, E3 +541085.340}
SPL {X  -162.820, Y  +613.536, Z    +0.000, E1   +22.242, E3 +541098.462}
SPL {X  -162.820, Y  +610.461, Z    +0.000, E1   +22.264, E3 +541114.093}
SPL {X  -162.820, Y  +607.796, Z    +0.000, E1   +22.261, E3 +541127.464}
SPL {X  -162.820, Y  +605.178, Z    +0.000, E1   +22.267, E3 +541140.948}
SPL {X  -162.820, Y  +602.350, Z    +0.000, E1   +22.224, E3 +541155.565}
SPL {X  -162.820, Y  +599.842, Z    +0.000, E1   +22.298, E3 +541167.716}
SPL {X  -162.820, Y  +597.194, Z    +0.000, E1   +22.253, E3 +541181.637}
SPL {X  -162.820, Y  +594.779, Z    +0.000, E1   +22.284, E3 +541193.541}
SPL {X  -162.820, Y  +593.320, Z    +0.000, E1   +22.199, E3 +541201.645}
SPL {X  -162.820, Y  +591.031, Z    +0.000, E1   +22.283, E3 +541212.736}
SPL {X  -162.820, Y  +588.026, Z    +0.000, E1   +22.301, E3 +541227.863}
SPL {X  -162.820, Y  +585.899, Z    +0.000, E1   +22.286, E3 +541238.665}
SPL {X  -162.820, Y  +583.204, Z    +0.000, E1   +22.278, E3 +541252.688}
SPL {X  -162.820, Y  +579.691, Z    +0.000, E1   +22.312, E3 +541270.176}
SPL {X  -162.820, Y  +577.460, Z    +0.000, E1   +22.218, E3 +541282.163}
SPL {X  -162.820, Y  +575.394, Z    +0.000, E1   +22.240, E3 +541292.588}
SPL {X  -162.820, Y  +572.645, Z    +0.000, E1   +22.246, E3 +541306.586}
SPL {X  -162.820, Y  +570.282, Z    +0.000, E1   +22.231, E3 +541318.636}
SPL {X  -162.820, Y  +567.961, Z    +0.000, E1   +22.247, E3 +541330.426}
SPL {X  -162.820, Y  +564.506, Z    +0.000, E1   +22.298, E3 +541347.740}
SPL {X  -162.820, Y  +561.620, Z    +0.000, E1   +22.191, E3 +541363.121}
SPL {X  -162.820, Y  +558.919, Z    +0.000, E1   +22.286, E3 +541376.167}
SPL {X  -162.820, Y  +555.548, Z    +0.000, E1   +22.322, E3 +541393.076}
SPL {X  -162.820, Y  +552.787, Z    +0.000, E1   +22.213, E3 +541407.874}
SPL {X  -162.820, Y  +550.136, Z    +0.000, E1   +22.258, E3 +541421.107}
SPL {X  -162.820, Y  +546.694, Z    +0.000, E1   +22.290, E3 +541438.429}
SPL {X  -162.820, Y  +543.558, Z    +0.000, E1   +22.285, E3 +541454.292}
SPL {X  -162.820, Y  +541.633, Z    +0.000, E1   +22.257, E3 +541464.220}
SPL {X  -162.820, Y  +539.116, Z    +0.000, E1   +22.302, E3 +541476.831}
SPL {X  -162.820, Y  +536.913, Z    +0.000, E1   +22.192, E3 +541488.756}
SPL {X  -162.820, Y  +534.880, Z    +0.000, E1   +22.252, E3 +541498.709}
SPL {X  -162.820, Y  +532.896, Z    +0.000, E1   +22.234, E3 +541508.869}
SPL {X  -162.820, Y  +531.056, Z    +0.000, E1   +22.251, E3 +541518.151}
SPL {X  -162.820, Y  +528.708, Z    +0.000, E1   +22.319, E3 +541529.533}
SPL {X  -162.820, Y  +525.932, Z    +0.000, E1   +22.258, E3 +541544.289}
SPL {X  -162.820, Y  +522.524, Z    +0.000, E1   +22.326, E3 +541561.013}
SPL {X  -162.820, Y  +519.457, Z    +0.000, E1   +22.481, E3 +541575.142}
SPL {X  -162.820, Y  +506.285, Z    +0.000, E1   +28.538, E3 +541586.600}
SPL {X  -162.820, Y  +504.441, Z    +0.000, E1   +27.574, E3 +541600.942}
SPL {X  -162.820, Y  +503.215, Z    +0.000, E1   +26.369, E3 +541614.449}
SPL {X  -162.820, Y  +502.265, Z    +0.000, E1   +25.287, E3 +541626.931}
SPL {X  -162.820, Y  +501.060, Z    +0.000, E1   +24.081, E3 +541641.672}
SPL {X  -162.820, Y  +500.336, Z    +0.000, E1   +23.110, E3 +541652.812}
SPL {X  -162.820, Y  +499.240, Z    +0.000, E1   +22.316, E3 +541665.122}
SPL {X  -162.820, Y  +498.027, Z    +0.000, E1   +21.516, E3 +541678.030}
SPL {X  -162.820, Y  +495.897, Z    +0.000, E1   +21.662, E3 +541687.950}
SPL {X  -162.820, Y  +493.717, Z    +0.000, E1   +21.704, E3 +541699.057}
SPL {X  -162.820, Y  +491.396, Z    +0.000, E1   +21.707, E3 +541711.181}
SPL {X  -162.820, Y  +488.560, Z    +0.000, E1   +21.695, E3 +541726.290}
SPL {X  -162.820, Y  +485.661, Z    +0.000, E1   +21.712, E3 +541741.175}
SPL {X  -162.820, Y  +483.668, Z    +0.000, E1   +21.664, E3 +541752.003}
SPL {X  -162.820, Y  +481.739, Z    +0.000, E1   +21.704, E3 +541761.717}
SPL {X  -162.820, Y  +479.894, Z    +0.000, E1   +21.695, E3 +541771.504}
SPL {X  -162.820, Y  +477.685, Z    +0.000, E1   +21.656, E3 +541783.441}
SPL {X  -162.820, Y  +475.419, Z    +0.000, E1   +21.711, E3 +541794.794}
SPL {X  -162.820, Y  +473.301, Z    +0.000, E1   +21.712, E3 +541805.891}
SPL {X  -162.820, Y  +470.965, Z    +0.000, E1   +21.700, E3 +541818.236}
SPL {X  -162.820, Y  +469.036, Z    +0.000, E1   +21.695, E3 +541828.280}
SPL {X  -162.820, Y  +467.138, Z    +0.000, E1   +21.678, E3 +541838.452}
SPL {X  -162.820, Y  +465.011, Z    +0.000, E1   +21.692, E3 +541849.434}
SPL {X  -162.820, Y  +462.669, Z    +0.000, E1   +21.752, E3 +541861.215}
SPL {X  -162.820, Y  +460.725, Z    +0.000, E1   +21.689, E3 +541871.828}
SPL {X  -162.820, Y  +458.666, Z    +0.000, E1   +21.695, E3 +541882.640}
SPL {X  -162.820, Y  +456.431, Z    +0.000, E1   +21.708, E3 +541894.168}
SPL {X  -162.820, Y  +454.628, Z    +0.000, E1   +21.674, E3 +541903.886}
SPL {X  -162.820, Y  +452.690, Z    +0.000, E1   +21.773, E3 +541913.160}
SPL {X  -162.820, Y  +450.610, Z    +0.000, E1   +21.698, E3 +541924.759}
SPL {X  -162.820, Y  +448.170, Z    +0.000, E1   +21.667, E3 +541937.780}
SPL {X  -162.820, Y  +446.246, Z    +0.000, E1   +21.696, E3 +541947.598}
SPL {X  -162.820, Y  +443.784, Z    +0.000, E1   +21.713, E3 +541960.384}
SPL {X  -162.820, Y  +440.567, Z    +0.000, E1   +21.731, E3 +541977.224}
SPL {X  -162.820, Y  +437.628, Z    +0.000, E1   +21.678, E3 +541992.888}
SPL {X  -162.820, Y  +435.262, Z    +0.000, E1   +21.727, E3 +542004.824}
SPL {X  -162.820, Y  +433.510, Z    +0.000, E1   +21.692, E3 +542014.237}
SPL {X  -162.820, Y  +431.492, Z    +0.000, E1   +21.686, E3 +542024.933}
SPL {X  -162.820, Y  +429.074, Z    +0.000, E1   +21.710, E3 +542037.385}
SPL {X  -162.820, Y  +426.023, Z    +0.000, E1   +21.718, E3 +542053.453}
SPL {X  -162.820, Y  +422.986, Z    +0.000, E1   +21.685, E3 +542069.500}
SPL {X  -162.820, Y  +420.528, Z    +0.000, E1   +21.706, E3 +542082.150}
SPL {X  -162.820, Y  +418.116, Z    +0.000, E1   +21.761, E3 +542094.297}
SPL {X  -162.820, Y  +416.127, Z    +0.000, E1   +21.715, E3 +542105.003}
SPL {X  -162.820, Y  +414.361, Z    +0.000, E1   +21.613, E3 +542115.190}
SPL {X  -162.820, Y  +411.450, Z    +0.000, E1   +21.710, E3 +542129.763}
SPL {X  -162.820, Y  +408.590, Z    +0.000, E1   +21.735, E3 +542144.389}
SPL {X  -162.820, Y  +406.238, Z    +0.000, E1   +21.697, E3 +542157.038}
SPL {X  -162.820, Y  +403.166, Z    +0.000, E1   +21.746, E3 +542172.844}
SPL {X  -162.820, Y  +400.348, Z    +0.000, E1   +21.713, E3 +542187.678}
SPL {X  -162.820, Y  +398.298, Z    +0.000, E1   +21.721, E3 +542198.294}
SPL {X  -162.820, Y  +396.371, Z    +0.000, E1   +21.713, E3 +542208.476}
SPL {X  -162.820, Y  +394.508, Z    +0.000, E1   +21.616, E3 +542219.031}
SPL {X  -162.820, Y  +391.777, Z    +0.000, E1   +21.714, E3 +542232.691}
SPL {X  -162.820, Y  +388.822, Z    +0.000, E1   +21.717, E3 +542248.010}
SPL {X  -162.820, Y  +386.818, Z    +0.000, E1   +21.679, E3 +542258.750}
SPL {X  -162.820, Y  +384.697, Z    +0.000, E1   +21.693, E3 +542269.821}
SPL {X  -162.820, Y  +382.288, Z    +0.000, E1   +21.742, E3 +542281.944}
SPL {X  -162.817, Y  +379.520, Z    +0.000, E1   +21.723, E3 +542296.782}
SPL {X  -162.776, Y  +376.710, Z    +0.000, E1   +21.698, E3 +542311.521}
SPL {X  -162.707, Y  +374.438, Z    +0.000, E1   +21.688, E3 +542323.525}
SPL {X  -162.607, Y  +372.171, Z    +0.000, E1   +21.692, E3 +542335.324}
SPL {X  -162.494, Y  +370.197, Z    +0.000, E1   +21.655, E3 +542345.950}
SPL {X  -162.349, Y  +368.131, Z    +0.000, E1   +21.624, E3 +542357.068}
SPL {X  -162.161, Y  +365.866, Z    +0.000, E1   +21.642, E3 +542368.754}
SPL {X  -161.651, Y  +361.024, Z    +0.000, E1   +22.970, E3 +542382.177}
SPL {X  -160.281, Y  +351.857, Z    +0.000, E1   +24.243, E3 +542417.516}
ENDSPLINE

SPLINE
SPL {X  -161.833, Y  +362.603, Z    +0.000, E1   +17.021, E3 +542432.212}
ENDSPLINE

SPLINE
SPL {X  -160.786, Y  +354.842, Z    +0.000, E1   +19.274, E3 +542464.367}
ENDSPLINE

SPLINE
SPL {X  -162.485, Y  +370.062, Z    +0.000, E1   +10.606, E3 +542470.746}
SPL {X  -162.820, Y  +381.311, Z    +0.000, E1    +4.054, E3 +542461.101}
SPL {X  -162.820, Y  +389.994, Z    +0.000, E1    -2.149, E3 +542455.513}
SPL {X  -162.820, Y  +391.982, Z    +0.000, E1    -3.443, E3 +542465.958}
SPL {X  -162.820, Y  +399.630, Z    +0.000, E1    -9.426, E3 +542468.466}
SPL {X  -162.820, Y  +408.127, Z    +0.000, E1   -18.417, E3 +542454.754}
SPL {X  -162.820, Y  +420.083, Z    +0.000, E1   -24.325, E3 +542475.230}
SPL {X  -162.820, Y  +428.527, Z    +0.000, E1   -26.988, E3 +542492.522}
SPL {X  -162.820, Y  +431.191, Z    +0.000, E1   -23.548, E3 +542527.375}
SPL {X  -162.820, Y  +432.946, Z    +0.000, E1   -22.795, E3 +542541.778}
SPL {X  -162.820, Y  +434.888, Z    +0.000, E1   -22.823, E3 +542551.185}
SPL {X  -162.820, Y  +436.834, Z    +0.000, E1   -22.779, E3 +542561.145}
SPL {X  -162.820, Y  +438.868, Z    +0.000, E1   -22.837, E3 +542570.799}
SPL {X  -162.820, Y  +441.351, Z    +0.000, E1   -22.805, E3 +542583.374}
SPL {X  -162.820, Y  +443.809, Z    +0.000, E1   -22.804, E3 +542595.540}
SPL {X  -162.820, Y  +447.077, Z    +0.000, E1   -22.869, E3 +542611.351}
SPL {X  -162.820, Y  +449.911, Z    +0.000, E1   -22.774, E3 +542625.960}
SPL {X  -162.820, Y  +451.861, Z    +0.000, E1   -22.750, E3 +542635.808}
SPL {X  -162.820, Y  +454.167, Z    +0.000, E1   -22.842, E3 +542646.537}
SPL {X  -162.820, Y  +456.529, Z    +0.000, E1   -22.855, E3 +542658.066}
SPL {X  -162.820, Y  +458.725, Z    +0.000, E1   -22.793, E3 +542669.470}
SPL {X  -162.820, Y  +460.754, Z    +0.000, E1   -22.806, E3 +542679.343}
SPL {X  -162.820, Y  +462.409, Z    +0.000, E1   -22.783, E3 +542687.760}
SPL {X  -162.820, Y  +464.633, Z    +0.000, E1   -22.813, E3 +542698.589}
SPL {X  -162.820, Y  +467.913, Z    +0.000, E1   -22.879, E3 +542714.428}
SPL {X  -162.820, Y  +470.892, Z    +0.000, E1   -22.837, E3 +542729.318}
SPL {X  -162.820, Y  +472.726, Z    +0.000, E1   -22.777, E3 +542738.856}
SPL {X  -162.820, Y  +475.118, Z    +0.000, E1   -22.777, E3 +542750.828}
SPL {X  -162.820, Y  +477.389, Z    +0.000, E1   -22.803, E3 +542761.744}
SPL {X  -162.820, Y  +478.914, Z    +0.000, E1   -22.821, E3 +542769.136}
SPL {X  -162.820, Y  +481.034, Z    +0.000, E1   -22.831, E3 +542779.658}
SPL {X  -162.820, Y  +484.256, Z    +0.000, E1   -22.840, E3 +542795.677}
SPL {X  -162.820, Y  +487.952, Z    +0.000, E1   -22.824, E3 +542814.107}
SPL {X  -162.820, Y  +490.653, Z    +0.000, E1   -22.810, E3 +542827.377}
SPL {X  -162.820, Y  +493.233, Z    +0.000, E1   -22.844, E3 +542840.055}
SPL {X  -162.820, Y  +496.150, Z    +0.000, E1   -22.796, E3 +542854.775}
SPL {X  -162.820, Y  +498.661, Z    +0.000, E1   -22.828, E3 +542866.955}
SPL {X  -162.820, Y  +501.761, Z    +0.000, E1   -22.820, E3 +542882.524}
SPL {X  -162.820, Y  +505.323, Z    +0.000, E1   -22.838, E3 +542899.971}
SPL {X  -162.820, Y  +507.875, Z    +0.000, E1   -22.849, E3 +542912.338}
SPL {X  -162.820, Y  +510.068, Z    +0.000, E1   -22.761, E3 +542924.031}
SPL {X  -162.820, Y  +512.359, Z    +0.000, E1   -22.823, E3 +542934.763}
SPL {X  -162.820, Y  +514.562, Z    +0.000, E1   -22.806, E3 +542945.949}
SPL {X  -162.820, Y  +517.952, Z    +0.000, E1   -22.864, E3 +542962.347}
SPL {X  -162.820, Y  +520.641, Z    +0.000, E1   -22.790, E3 +542976.065}
SPL {X  -162.820, Y  +522.740, Z    +0.000, E1   -22.811, E3 +542986.308}
SPL {X  -162.820, Y  +524.628, Z    +0.000, E1   -22.846, E3 +542995.303}
SPL {X  -162.820, Y  +526.661, Z    +0.000, E1   -22.801, E3 +543005.858}
SPL {X  -162.820, Y  +529.662, Z    +0.000, E1   -22.810, E3 +543020.709}
SPL {X  -162.820, Y  +532.614, Z    +0.000, E1   -22.828, E3 +543035.115}
SPL {X  -162.820, Y  +534.838, Z    +0.000, E1   -22.864, E3 +543045.744}
SPL {X  -162.820, Y  +536.882, Z    +0.000, E1   -22.782, E3 +543056.599}
SPL {X  -162.820, Y  +539.194, Z    +0.000, E1   -22.826, E3 +543067.647}
SPL {X  -162.820, Y  +541.555, Z    +0.000, E1   -22.817, E3 +543079.462}
SPL {X  -162.820, Y  +543.728, Z    +0.000, E1   -22.799, E3 +543090.319}
SPL {X  -162.820, Y  +545.925, Z    +0.000, E1   -22.803, E3 +543101.189}
SPL {X  -162.820, Y  +548.328, Z    +0.000, E1   -22.796, E3 +543113.185}
SPL {X  -162.820, Y  +551.027, Z    +0.000, E1   -22.819, E3 +543126.378}
SPL {X  -162.820, Y  +553.721, Z    +0.000, E1   -22.807, E3 +543139.822}
SPL {X  -162.820, Y  +556.430, Z    +0.000, E1   -22.821, E3 +543153.118}
SPL {X  -162.820, Y  +559.675, Z    +0.000, E1   -22.837, E3 +543169.198}
SPL {X  -162.820, Y  +562.799, Z    +0.000, E1   -22.814, E3 +543184.704}
SPL {X  -162.820, Y  +565.170, Z    +0.000, E1   -22.801, E3 +543196.529}
SPL {X  -162.820, Y  +568.020, Z    +0.000, E1   -22.787, E3 +543210.916}
SPL {X  -162.820, Y  +570.992, Z    +0.000, E1   -22.834, E3 +543225.135}
SPL {X  -162.820, Y  +572.901, Z    +0.000, E1   -22.775, E3 +543235.003}
SPL {X  -162.820, Y  +575.638, Z    +0.000, E1   -22.855, E3 +543248.113}
SPL {X  -162.820, Y  +578.553, Z    +0.000, E1   -22.801, E3 +543262.825}
SPL {X  -162.820, Y  +581.064, Z    +0.000, E1   -22.823, E3 +543275.110}
SPL {X  -162.820, Y  +583.435, Z    +0.000, E1   -22.808, E3 +543286.931}
SPL {X  -162.820, Y  +585.410, Z    +0.000, E1   -22.764, E3 +543297.067}
SPL {X  -162.820, Y  +587.676, Z    +0.000, E1   -22.853, E3 +543307.582}
SPL {X  -162.820, Y  +589.682, Z    +0.000, E1   -22.776, E3 +543318.112}
SPL {X  -162.820, Y  +591.720, Z    +0.000, E1   -22.868, E3 +543327.422}
SPL {X  -162.820, Y  +593.650, Z    +0.000, E1   -22.810, E3 +543337.492}
SPL {X  -162.820, Y  +595.830, Z    +0.000, E1   -22.828, E3 +543348.108}
SPL {X  -162.820, Y  +598.094, Z    +0.000, E1   -22.843, E3 +543359.221}
SPL {X  -162.820, Y  +600.420, Z    +0.000, E1   -22.826, E3 +543370.852}
SPL {X  -162.820, Y  +602.573, Z    +0.000, E1   -22.830, E3 +543381.438}
SPL {X  -162.820, Y  +604.828, Z    +0.000, E1   -22.784, E3 +543393.076}
SPL {X  -162.820, Y  +607.142, Z    +0.000, E1   -22.808, E3 +543404.257}
SPL {X  -162.820, Y  +608.890, Z    +0.000, E1   -22.790, E3 +543413.081}
SPL {X  -162.820, Y  +611.103, Z    +0.000, E1   -22.785, E3 +543424.119}
SPL {X  -162.820, Y  +613.294, Z    +0.000, E1   -22.780, E3 +543434.993}
SPL {X  -162.820, Y  +615.356, Z    +0.000, E1   -22.799, E3 +543445.050}
SPL {X  -162.820, Y  +617.439, Z    +0.000, E1   -22.808, E3 +543455.308}
SPL {X  -162.820, Y  +619.665, Z    +0.000, E1   -22.817, E3 +543466.276}
SPL {X  -162.820, Y  +621.733, Z    +0.000, E1   -22.759, E3 +543477.000}
SPL {X  -162.820, Y  +624.076, Z    +0.000, E1   -22.774, E3 +543488.505}
SPL {X  -162.820, Y  +626.527, Z    +0.000, E1   -22.768, E3 +543500.748}
SPL {X  -162.820, Y  +629.758, Z    +0.000, E1   -22.800, E3 +543516.677}
SPL {X  -162.820, Y  +632.572, Z    +0.000, E1   -22.785, E3 +543530.526}
SPL {X  -162.820, Y  +634.507, Z    +0.000, E1   -22.784, E3 +543540.165}
SPL {X  -162.820, Y  +636.863, Z    +0.000, E1   -22.760, E3 +543552.087}
SPL {X  -162.820, Y  +639.254, Z    +0.000, E1   -22.767, E3 +543563.870}
SPL {X  -162.820, Y  +641.195, Z    +0.000, E1   -22.782, E3 +543573.318}
SPL {X  -162.820, Y  +643.449, Z    +0.000, E1   -22.796, E3 +543584.488}
SPL {X  -162.820, Y  +645.630, Z    +0.000, E1   -22.795, E3 +543595.184}
SPL {X  -162.820, Y  +647.561, Z    +0.000, E1   -22.705, E3 +543605.634}
SPL {X  -162.820, Y  +651.051, Z    +0.000, E1   -22.833, E3 +543622.054}
SPL {X  -162.820, Y  +653.898, Z    +0.000, E1   -22.796, E3 +543636.240}
SPL {X  -162.820, Y  +656.161, Z    +0.000, E1   -22.812, E3 +543647.361}
SPL {X  -162.820, Y  +658.384, Z    +0.000, E1   -22.822, E3 +543658.227}
SPL {X  -162.820, Y  +660.215, Z    +0.000, E1   -22.649, E3 +543668.818}
SPL {X  -162.820, Y  +662.823, Z    +0.000, E1   -22.799, E3 +543680.526}
SPL {X  -162.820, Y  +665.112, Z    +0.000, E1   -22.835, E3 +543691.580}
SPL {X  -162.820, Y  +667.016, Z    +0.000, E1   -22.823, E3 +543701.009}
SPL {X  -162.820, Y  +668.960, Z    +0.000, E1   -22.773, E3 +543711.176}
SPL {X  -162.820, Y  +672.333, Z    +0.000, E1   -22.837, E3 +543727.512}
SPL {X  -162.812, Y  +675.071, Z    +0.000, E1   -22.742, E3 +543741.657}
SPL {X  -162.773, Y  +677.428, Z    +0.000, E1   -22.762, E3 +543753.255}
SPL {X  -162.691, Y  +679.987, Z    +0.000, E1   -22.794, E3 +543765.668}
SPL {X  -162.604, Y  +681.880, Z    +0.000, E1   -22.691, E3 +543775.829}
SPL {X  -162.458, Y  +684.346, Z    +0.000, E1   -22.764, E3 +543787.623}
SPL {X  -162.296, Y  +686.547, Z    +0.000, E1   -22.660, E3 +543799.239}
SPL {X  -162.090, Y  +688.902, Z    +0.000, E1   -22.700, E3 +543810.748}
SPL {X  -161.474, Y  +694.390, Z    +0.000, E1   -24.298, E3 +543824.103}
SPL {X  -158.553, Y  +710.529, Z    +0.000, E1   -30.890, E3 +543840.665}
ENDSPLINE

SPLINE
SPL {X  -161.215, Y  +696.305, Z    +0.000, E1   -20.575, E3 +543867.245}
SPL {X  -161.691, Y  +692.643, Z    +0.000, E1   -17.369, E3 +543883.434}
SPL {X  -162.534, Y  +683.153, Z    +0.000, E1   -10.475, E3 +543908.901}
SPL {X  -162.820, Y  +667.630, Z    +0.000, E1    -0.882, E3 +543902.877}
SPL {X  -162.820, Y  +661.883, Z    +0.000, E1    +3.373, E3 +543908.320}
SPL {X  -162.820, Y  +653.808, Z    +0.000, E1    +9.891, E3 +543906.011}
SPL {X  -162.820, Y  +632.548, Z    +0.000, E1   +27.446, E3 +543902.548}
ENDSPLINE

SPLINE
SPL {X  -162.820, Y  +638.080, Z    +0.000, E1   +18.858, E3 +543930.297}
ENDSPLINE

SPLINE
SPL {X  -162.820, Y  +623.278, Z    +0.000, E1   +28.723, E3 +543931.867}
SPL {X  -162.820, Y  +618.658, Z    +0.000, E1   +26.841, E3 +543960.476}
ENDSPLINE

SPLINE
SPL {X  -162.820, Y  +623.685, Z    +0.000, E1   +22.346, E3 +543972.783}
ENDSPLINE

SPLINE
SPL {X  -162.820, Y  +621.304, Z    +0.000, E1   +22.259, E3 +543985.598}
SPL {X  -162.820, Y  +618.758, Z    +0.000, E1   +22.239, E3 +543998.749}
SPL {X  -162.820, Y  +616.062, Z    +0.000, E1   +22.275, E3 +544012.169}
SPL {X  -162.820, Y  +613.536, Z    +0.000, E1   +22.242, E3 +544025.291}
SPL {X  -162.820, Y  +610.461, Z    +0.000, E1   +22.264, E3 +544040.922}
SPL {X  -162.820, Y  +606.755, Z    +0.000, E1   +22.275, E3 +544059.720}
SPL {X  -162.820, Y  +603.020, Z    +0.000, E1   +22.272, E3 +544078.780}
SPL {X  -162.820, Y  +599.168, Z    +0.000, E1   +22.310, E3 +544098.048}
SPL {X  -162.820, Y  +596.569, Z    +0.000, E1   +22.222, E3 +544111.770}
SPL {X  -162.820, Y  +594.115, Z    +0.000, E1   +22.273, E3 +544123.996}
SPL {X  -162.820, Y  +591.721, Z    +0.000, E1   +22.239, E3 +544136.311}
SPL {X  -162.820, Y  +589.492, Z    +0.000, E1   +22.304, E3 +544147.172}
SPL {X  -162.820, Y  +587.447, Z    +0.000, E1   +22.279, E3 +544157.701}
SPL {X  -162.820, Y  +585.192, Z    +0.000, E1   +22.298, E3 +544169.111}
SPL {X  -162.820, Y  +582.610, Z    +0.000, E1   +22.234, E3 +544182.734}
SPL {X  -162.820, Y  +580.317, Z    +0.000, E1   +22.300, E3 +544193.788}
SPL {X  -162.820, Y  +578.878, Z    +0.000, E1   +22.272, E3 +544201.297}
SPL {X  -162.820, Y  +576.856, Z    +0.000, E1   +22.233, E3 +544212.056}
SPL {X  -162.820, Y  +573.830, Z    +0.000, E1   +22.272, E3 +544227.192}
SPL {X  -162.820, Y  +570.852, Z    +0.000, E1   +22.234, E3 +544242.651}
SPL {X  -162.820, Y  +568.608, Z    +0.000, E1   +22.253, E3 +544253.785}
SPL {X  -162.820, Y  +565.838, Z    +0.000, E1   +22.271, E3 +544268.016}
SPL {X  -162.820, Y  +562.162, Z    +0.000, E1   +22.252, E3 +544286.833}
SPL {X  -162.820, Y  +558.919, Z    +0.000, E1   +22.286, E3 +544302.996}
SPL {X  -162.820, Y  +555.548, Z    +0.000, E1   +22.322, E3 +544319.905}
SPL {X  -162.820, Y  +552.787, Z    +0.000, E1   +22.213, E3 +544334.703}
SPL {X  -162.820, Y  +550.871, Z    +0.000, E1   +22.229, E3 +544344.297}
SPL {X  -162.820, Y  +548.168, Z    +0.000, E1   +22.298, E3 +544357.634}
SPL {X  -162.820, Y  +545.860, Z    +0.000, E1   +22.216, E3 +544369.891}
SPL {X  -162.820, Y  +543.558, Z    +0.000, E1   +22.285, E3 +544381.122}
SPL {X  -162.820, Y  +540.968, Z    +0.000, E1   +22.274, E3 +544394.394}
SPL {X  -162.820, Y  +537.857, Z    +0.000, E1   +22.280, E3 +544410.270}
SPL {X  -162.820, Y  +534.880, Z    +0.000, E1   +22.252, E3 +544425.538}
SPL {X  -162.820, Y  +532.896, Z    +0.000, E1   +22.234, E3 +544435.699}
SPL {X  -162.820, Y  +531.056, Z    +0.000, E1   +22.251, E3 +544444.981}
SPL {X  -162.820, Y  +528.708, Z    +0.000, E1   +22.319, E3 +544456.362}
SPL {X  -162.820, Y  +525.932, Z    +0.000, E1   +22.258, E3 +544471.118}
SPL {X  -162.820, Y  +522.524, Z    +0.000, E1   +22.326, E3 +544487.842}
SPL {X  -162.820, Y  +519.457, Z    +0.000, E1   +22.481, E3 +544501.971}
SPL {X  -162.820, Y  +506.285, Z    +0.000, E1   +28.538, E3 +544513.429}
SPL {X  -162.820, Y  +504.441, Z    +0.000, E1   +27.574, E3 +544527.771}
SPL {X  -162.820, Y  +502.813, Z    +0.000, E1   +26.013, E3 +544545.969}
SPL {X  -162.820, Y  +502.016, Z    +0.000, E1   +24.802, E3 +544558.312}
SPL {X  -162.820, Y  +501.060, Z    +0.000, E1   +24.081, E3 +544568.501}
SPL {X  -162.820, Y  +500.336, Z    +0.000, E1   +23.110, E3 +544579.641}
SPL {X  -162.820, Y  +499.240, Z    +0.000, E1   +22.316, E3 +544591.952}
SPL {X  -162.820, Y  +498.027, Z    +0.000, E1   +21.516, E3 +544604.859}
SPL {X  -162.820, Y  +495.897, Z    +0.000, E1   +21.662, E3 +544614.780}
SPL {X  -162.820, Y  +493.717, Z    +0.000, E1   +21.704, E3 +544625.886}
SPL {X  -162.820, Y  +491.396, Z    +0.000, E1   +21.707, E3 +544638.010}
SPL {X  -162.820, Y  +488.560, Z    +0.000, E1   +21.695, E3 +544653.119}
SPL {X  -162.820, Y  +485.661, Z    +0.000, E1   +21.712, E3 +544668.005}
SPL {X  -162.820, Y  +483.668, Z    +0.000, E1   +21.664, E3 +544678.832}
SPL {X  -162.820, Y  +481.739, Z    +0.000, E1   +21.704, E3 +544688.546}
SPL {X  -162.820, Y  +479.894, Z    +0.000, E1   +21.695, E3 +544698.333}
SPL {X  -162.820, Y  +477.685, Z    +0.000, E1   +21.656, E3 +544710.271}
SPL {X  -162.820, Y  +475.419, Z    +0.000, E1   +21.711, E3 +544721.623}
SPL {X  -162.820, Y  +473.301, Z    +0.000, E1   +21.712, E3 +544732.721}
SPL {X  -162.820, Y  +470.965, Z    +0.000, E1   +21.700, E3 +544745.065}
SPL {X  -162.820, Y  +469.036, Z    +0.000, E1   +21.695, E3 +544755.109}
SPL {X  -162.820, Y  +467.138, Z    +0.000, E1   +21.678, E3 +544765.281}
SPL {X  -162.820, Y  +465.011, Z    +0.000, E1   +21.692, E3 +544776.263}
SPL {X  -162.820, Y  +462.669, Z    +0.000, E1   +21.752, E3 +544788.044}
SPL {X  -162.820, Y  +460.725, Z    +0.000, E1   +21.689, E3 +544798.657}
SPL {X  -162.820, Y  +458.666, Z    +0.000, E1   +21.695, E3 +544809.469}
SPL {X  -162.820, Y  +456.431, Z    +0.000, E1   +21.708, E3 +544820.997}
SPL {X  -162.820, Y  +454.628, Z    +0.000, E1   +21.674, E3 +544830.716}
SPL {X  -162.820, Y  +452.690, Z    +0.000, E1   +21.773, E3 +544839.990}
SPL {X  -162.820, Y  +450.610, Z    +0.000, E1   +21.698, E3 +544851.589}
SPL {X  -162.820, Y  +448.170, Z    +0.000, E1   +21.667, E3 +544864.609}
SPL {X  -162.820, Y  +446.246, Z    +0.000, E1   +21.696, E3 +544874.427}
SPL {X  -162.820, Y  +443.784, Z    +0.000, E1   +21.713, E3 +544887.213}
SPL {X  -162.820, Y  +441.754, Z    +0.000, E1   +21.708, E3 +544897.765}
SPL {X  -162.820, Y  +439.933, Z    +0.000, E1   +21.690, E3 +544907.529}
SPL {X  -162.820, Y  +437.628, Z    +0.000, E1   +21.678, E3 +544919.717}
SPL {X  -162.820, Y  +434.473, Z    +0.000, E1   +21.747, E3 +544935.813}
SPL {X  -162.820, Y  +431.492, Z    +0.000, E1   +21.686, E3 +544951.762}
SPL {X  -162.820, Y  +429.074, Z    +0.000, E1   +21.710, E3 +544964.214}
SPL {X  -162.820, Y  +426.023, Z    +0.000, E1   +21.718, E3 +544980.282}
SPL {X  -162.820, Y  +422.986, Z    +0.000, E1   +21.685, E3 +544996.329}
SPL {X  -162.820, Y  +420.528, Z    +0.000, E1   +21.706, E3 +545008.979}
SPL {X  -162.820, Y  +418.116, Z    +0.000, E1   +21.761, E3 +545021.127}
SPL {X  -162.820, Y  +416.127, Z    +0.000, E1   +21.715, E3 +545031.832}
SPL {X  -162.820, Y  +414.361, Z    +0.000, E1   +21.613, E3 +545042.019}
SPL {X  -162.820, Y  +411.450, Z    +0.000, E1   +21.710, E3 +545056.593}
SPL {X  -162.820, Y  +408.590, Z    +0.000, E1   +21.735, E3 +545071.218}
SPL {X  -162.820, Y  +406.238, Z    +0.000, E1   +21.697, E3 +545083.867}
SPL {X  -162.820, Y  +403.166, Z    +0.000, E1   +21.746, E3 +545099.673}
SPL {X  -162.820, Y  +400.348, Z    +0.000, E1   +21.713, E3 +545114.508}
SPL {X  -162.820, Y  +398.298, Z    +0.000, E1   +21.721, E3 +545125.123}
SPL {X  -162.820, Y  +396.371, Z    +0.000, E1   +21.713, E3 +545135.305}
SPL {X  -162.820, Y  +394.508, Z    +0.000, E1   +21.616, E3 +545145.861}
SPL {X  -162.820, Y  +392.435, Z    +0.000, E1   +21.681, E3 +545156.214}
SPL {X  -162.820, Y  +389.390, Z    +0.000, E1   +21.742, E3 +545171.821}
SPL {X  -162.820, Y  +386.818, Z    +0.000, E1   +21.679, E3 +545185.579}
SPL {X  -162.820, Y  +384.697, Z    +0.000, E1   +21.693, E3 +545196.650}
SPL {X  -162.820, Y  +382.288, Z    +0.000, E1   +21.742, E3 +545208.773}
SPL {X  -162.817, Y  +379.520, Z    +0.000, E1   +21.723, E3 +545223.611}
SPL {X  -162.776, Y  +376.710, Z    +0.000, E1   +21.698, E3 +545238.350}
SPL {X  -162.707, Y  +374.438, Z    +0.000, E1   +21.688, E3 +545250.354}
SPL {X  -162.607, Y  +372.171, Z    +0.000, E1   +21.692, E3 +545262.153}
SPL {X  -162.494, Y  +370.197, Z    +0.000, E1   +21.655, E3 +545272.780}
SPL {X  -162.349, Y  +368.131, Z    +0.000, E1   +21.624, E3 +545283.898}
SPL {X  -162.161, Y  +365.866, Z    +0.000, E1   +21.642, E3 +545295.583}
SPL {X  -161.651, Y  +361.024, Z    +0.000, E1   +22.970, E3 +545309.006}
SPL {X  -160.281, Y  +351.857, Z    +0.000, E1   +24.243, E3 +545344.345}
ENDSPLINE

SPLINE
SPL {X  -161.833, Y  +362.603, Z    +0.000, E1   +17.021, E3 +545359.041}
ENDSPLINE

SPLINE
SPL {X  -160.786, Y  +354.842, Z    +0.000, E1   +19.274, E3 +545391.197}
ENDSPLINE

SPLINE
SPL {X  -162.485, Y  +370.062, Z    +0.000, E1   +10.606, E3 +545397.575}
SPL {X  -162.818, Y  +379.636, Z    +0.000, E1    +5.115, E3 +545386.924}
SPL {X  -162.820, Y  +386.976, Z    +0.000, E1    +0.144, E3 +545386.023}
SPL {X  -162.820, Y  +391.982, Z    +0.000, E1    -3.443, E3 +545392.788}
SPL {X  -162.820, Y  +399.630, Z    +0.000, E1    -9.426, E3 +545395.295}
SPL {X  -162.820, Y  +408.127, Z    +0.000, E1   -18.417, E3 +545381.584}
SPL {X  -162.820, Y  +420.083, Z    +0.000, E1   -24.325, E3 +545402.059}
SPL {X  -162.820, Y  +428.527, Z    +0.000, E1   -26.988, E3 +545419.351}
SPL {X  -162.820, Y  +431.336, Z    +0.000, E1   -24.162, E3 +545449.561}
SPL {X  -162.820, Y  +432.048, Z    +0.000, E1   -22.832, E3 +545464.065}
SPL {X  -162.820, Y  +434.888, Z    +0.000, E1   -22.823, E3 +545478.014}
SPL {X  -162.820, Y  +436.834, Z    +0.000, E1   -22.779, E3 +545487.974}
SPL {X  -162.820, Y  +438.868, Z    +0.000, E1   -22.837, E3 +545497.628}
SPL {X  -162.820, Y  +441.351, Z    +0.000, E1   -22.805, E3 +545510.203}
SPL {X  -162.820, Y  +443.809, Z    +0.000, E1   -22.804, E3 +545522.370}
SPL {X  -162.820, Y  +446.105, Z    +0.000, E1   -22.815, E3 +545533.612}
SPL {X  -162.820, Y  +447.974, Z    +0.000, E1   -22.856, E3 +545542.515}
SPL {X  -162.820, Y  +449.911, Z    +0.000, E1   -22.774, E3 +545552.789}
SPL {X  -162.820, Y  +451.861, Z    +0.000, E1   -22.750, E3 +545562.637}
SPL {X  -162.820, Y  +454.167, Z    +0.000, E1   -22.842, E3 +545573.366}
SPL {X  -162.820, Y  +456.529, Z    +0.000, E1   -22.855, E3 +545584.895}
SPL {X  -162.820, Y  +458.725, Z    +0.000, E1   -22.793, E3 +545596.299}
SPL {X  -162.820, Y  +461.700, Z    +0.000, E1   -22.822, E3 +545610.922}
SPL {X  -162.820, Y  +464.633, Z    +0.000, E1   -22.813, E3 +545625.418}
SPL {X  -162.820, Y  +466.699, Z    +0.000, E1   -22.824, E3 +545635.465}
SPL {X  -162.820, Y  +468.655, Z    +0.000, E1   -22.858, E3 +545644.908}
SPL {X  -162.820, Y  +470.892, Z    +0.000, E1   -22.837, E3 +545656.147}
SPL {X  -162.820, Y  +473.485, Z    +0.000, E1   -22.806, E3 +545669.345}
SPL {X  -162.820, Y  +476.589, Z    +0.000, E1   -22.788, E3 +545684.867}
SPL {X  -162.820, Y  +478.914, Z    +0.000, E1   -22.821, E3 +545695.965}
SPL {X  -162.820, Y  +481.034, Z    +0.000, E1   -22.831, E3 +545706.487}
SPL {X  -162.820, Y  +484.256, Z    +0.000, E1   -22.840, E3 +545722.506}
SPL {X  -162.820, Y  +487.014, Z    +0.000, E1   -22.789, E3 +545736.373}
SPL {X  -162.820, Y  +489.750, Z    +0.000, E1   -22.832, E3 +545749.747}
SPL {X  -162.820, Y  +493.233, Z    +0.000, E1   -22.844, E3 +545766.884}
SPL {X  -162.820, Y  +496.150, Z    +0.000, E1   -22.796, E3 +545781.604}
SPL {X  -162.820, Y  +498.661, Z    +0.000, E1   -22.828, E3 +545793.785}
SPL {X  -162.820, Y  +501.761, Z    +0.000, E1   -22.820, E3 +545809.353}
SPL {X  -162.820, Y  +505.323, Z    +0.000, E1   -22.838, E3 +545826.800}
SPL {X  -162.820, Y  +507.875, Z    +0.000, E1   -22.849, E3 +545839.167}
SPL {X  -162.820, Y  +510.068, Z    +0.000, E1   -22.761, E3 +545850.860}
SPL {X  -162.820, Y  +512.359, Z    +0.000, E1   -22.823, E3 +545861.592}
SPL {X  -162.820, Y  +514.562, Z    +0.000, E1   -22.806, E3 +545872.779}
SPL {X  -162.820, Y  +517.952, Z    +0.000, E1   -22.864, E3 +545889.176}
SPL {X  -162.820, Y  +520.641, Z    +0.000, E1   -22.790, E3 +545902.895}
SPL {X  -162.820, Y  +522.740, Z    +0.000, E1   -22.811, E3 +545913.137}
SPL {X  -162.820, Y  +524.628, Z    +0.000, E1   -22.846, E3 +545922.132}
SPL {X  -162.820, Y  +526.661, Z    +0.000, E1   -22.801, E3 +545932.688}
SPL {X  -162.820, Y  +529.662, Z    +0.000, E1   -22.810, E3 +545947.538}
SPL {X  -162.820, Y  +532.614, Z    +0.000, E1   -22.828, E3 +545961.945}
SPL {X  -162.820, Y  +534.838, Z    +0.000, E1   -22.864, E3 +545972.573}
SPL {X  -162.820, Y  +536.882, Z    +0.000, E1   -22.782, E3 +545983.428}
SPL {X  -162.820, Y  +539.194, Z    +0.000, E1   -22.826, E3 +545994.477}
SPL {X  -162.820, Y  +541.555, Z    +0.000, E1   -22.817, E3 +546006.291}
SPL {X  -162.820, Y  +543.728, Z    +0.000, E1   -22.799, E3 +546017.149}
SPL {X  -162.820, Y  +545.925, Z    +0.000, E1   -22.803, E3 +546028.019}
SPL {X  -162.820, Y  +549.071, Z    +0.000, E1   -22.836, E3 +546043.546}
SPL {X  -162.820, Y  +553.089, Z    +0.000, E1   -22.838, E3 +546063.446}
SPL {X  -162.820, Y  +556.430, Z    +0.000, E1   -22.821, E3 +546079.947}
SPL {X  -162.820, Y  +558.974, Z    +0.000, E1   -22.806, E3 +546092.647}
SPL {X  -162.820, Y  +562.171, Z    +0.000, E1   -22.845, E3 +546108.345}
SPL {X  -162.820, Y  +565.170, Z    +0.000, E1   -22.801, E3 +546123.358}
SPL {X  -162.820, Y  +567.308, Z    +0.000, E1   -22.750, E3 +546134.375}
SPL {X  -162.820, Y  +570.378, Z    +0.000, E1   -22.843, E3 +546148.998}
SPL {X  -162.820, Y  +573.634, Z    +0.000, E1   -22.827, E3 +546165.142}
SPL {X  -162.820, Y  +576.228, Z    +0.000, E1   -22.814, E3 +546178.039}
SPL {X  -162.820, Y  +578.553, Z    +0.000, E1   -22.801, E3 +546189.654}
SPL {X  -162.820, Y  +581.064, Z    +0.000, E1   -22.823, E3 +546201.939}
SPL {X  -162.820, Y  +583.435, Z    +0.000, E1   -22.808, E3 +546213.761}
SPL {X  -162.820, Y  +585.410, Z    +0.000, E1   -22.764, E3 +546223.896}
SPL {X  -162.820, Y  +587.676, Z    +0.000, E1   -22.853, E3 +546234.411}
SPL {X  -162.820, Y  +590.707, Z    +0.000, E1   -22.855, E3 +546249.561}
SPL {X  -162.820, Y  +593.650, Z    +0.000, E1   -22.810, E3 +546264.321}
SPL {X  -162.820, Y  +595.830, Z    +0.000, E1   -22.828, E3 +546274.937}
SPL {X  -162.820, Y  +598.094, Z    +0.000, E1   -22.843, E3 +546286.050}
SPL {X  -162.820, Y  +600.420, Z    +0.000, E1   -22.826, E3 +546297.682}
SPL {X  -162.820, Y  +603.245, Z    +0.000, E1   -22.831, E3 +546311.747}
SPL {X  -162.820, Y  +606.456, Z    +0.000, E1   -22.811, E3 +546327.792}
SPL {X  -162.820, Y  +608.890, Z    +0.000, E1   -22.790, E3 +546339.910}
SPL {X  -162.820, Y  +611.103, Z    +0.000, E1   -22.785, E3 +546350.949}
SPL {X  -162.820, Y  +613.294, Z    +0.000, E1   -22.780, E3 +546361.822}
SPL {X  -162.820, Y  +615.356, Z    +0.000, E1   -22.799, E3 +546371.879}
SPL {X  -162.820, Y  +617.439, Z    +0.000, E1   -22.808, E3 +546382.137}
SPL {X  -162.820, Y  +619.665, Z    +0.000, E1   -22.817, E3 +546393.105}
SPL {X  -162.820, Y  +621.733, Z    +0.000, E1   -22.759, E3 +546403.829}
SPL {X  -162.820, Y  +624.076, Z    +0.000, E1   -22.774, E3 +546415.335}
SPL {X  -162.820, Y  +627.244, Z    +0.000, E1   -22.803, E3 +546431.017}
SPL {X  -162.820, Y  +630.349, Z    +0.000, E1   -22.766, E3 +546446.549}
SPL {X  -162.820, Y  +632.572, Z    +0.000, E1   -22.785, E3 +546457.355}
SPL {X  -162.820, Y  +634.507, Z    +0.000, E1   -22.784, E3 +546466.994}
SPL {X  -162.820, Y  +636.863, Z    +0.000, E1   -22.760, E3 +546478.916}
SPL {X  -162.820, Y  +640.111, Z    +0.000, E1   -22.809, E3 +546494.799}
SPL {X  -162.820, Y  +643.449, Z    +0.000, E1   -22.796, E3 +546511.317}
SPL {X  -162.820, Y  +645.630, Z    +0.000, E1   -22.795, E3 +546522.013}
SPL {X  -162.820, Y  +647.561, Z    +0.000, E1   -22.705, E3 +546532.464}
SPL {X  -162.820, Y  +649.758, Z    +0.000, E1   -22.780, E3 +546542.654}
SPL {X  -162.820, Y  +651.708, Z    +0.000, E1   -22.810, E3 +546552.148}
SPL {X  -162.820, Y  +653.898, Z    +0.000, E1   -22.796, E3 +546563.069}
SPL {X  -162.820, Y  +656.161, Z    +0.000, E1   -22.812, E3 +546574.190}
SPL {X  -162.820, Y  +658.384, Z    +0.000, E1   -22.822, E3 +546585.057}
SPL {X  -162.820, Y  +660.215, Z    +0.000, E1   -22.649, E3 +546595.647}
SPL {X  -162.820, Y  +662.823, Z    +0.000, E1   -22.799, E3 +546607.355}
SPL {X  -162.820, Y  +665.112, Z    +0.000, E1   -22.835, E3 +546618.410}
SPL {X  -162.820, Y  +667.016, Z    +0.000, E1   -22.823, E3 +546627.838}
SPL {X  -162.820, Y  +668.960, Z    +0.000, E1   -22.773, E3 +546638.006}
SPL {X  -162.820, Y  +672.333, Z    +0.000, E1   -22.837, E3 +546654.341}
SPL {X  -162.812, Y  +675.071, Z    +0.000, E1   -22.742, E3 +546668.487}
SPL {X  -162.773, Y  +677.428, Z    +0.000, E1   -22.762, E3 +546680.084}
SPL {X  -162.691, Y  +679.987, Z    +0.000, E1   -22.794, E3 +546692.497}
SPL {X  -162.604, Y  +681.880, Z    +0.000, E1   -22.691, E3 +546702.658}
SPL {X  -162.458, Y  +684.346, Z    +0.000, E1   -22.764, E3 +546714.452}
SPL {X  -162.296, Y  +686.547, Z    +0.000, E1   -22.660, E3 +546726.069}
SPL {X  -162.164, Y  +688.106, Z    +0.000, E1   -22.661, E3 +546733.802}
SPL {X  -161.938, Y  +690.422, Z    +0.000, E1   -22.769, E3 +546744.478}
SPL {X  -161.065, Y  +697.344, Z    +0.000, E1   -25.698, E3 +546753.597}
SPL {X  -158.730, Y  +709.763, Z    +0.000, E1   -31.225, E3 +546762.271}
ENDSPLINE

SPLINE
SPL {X  -160.932, Y  +698.225, Z    +0.000, E1   -21.712, E3 +546793.380}
SPL {X  -161.917, Y  +690.622, Z    +0.000, E1   -16.445, E3 +546806.981}
ENDSPLINE

SPLINE
SPL {X  -161.349, Y  +695.340, Z    +0.000, E1   -18.625, E3 +546814.599}
ENDSPLINE

SPLINE
SPL {X  -162.534, Y  +683.153, Z    +0.000, E1   -10.475, E3 +546835.730}
SPL {X  -162.820, Y  +667.630, Z    +0.000, E1    -0.882, E3 +546829.706}
SPL {X  -162.820, Y  +661.883, Z    +0.000, E1    +3.373, E3 +546835.149}
SPL {X  -162.820, Y  +655.163, Z    +0.000, E1    +8.702, E3 +546834.748}
SPL {X  -162.820, Y  +634.515, Z    +0.000, E1   +26.439, E3 +546827.161}
ENDSPLINE

SPLINE
SPL {X  -162.820, Y  +638.080, Z    +0.000, E1   +18.858, E3 +546857.126}
ENDSPLINE

SPLINE
SPL {X  -162.820, Y  +623.278, Z    +0.000, E1   +28.723, E3 +546858.696}
SPL {X  -162.820, Y  +618.658, Z    +0.000, E1   +26.841, E3 +546887.305}
ENDSPLINE

SPLINE
SPL {X  -162.820, Y  +623.685, Z    +0.000, E1   +22.346, E3 +546899.612}
ENDSPLINE

SPLINE
SPL {X  -162.820, Y  +621.304, Z    +0.000, E1   +22.259, E3 +546912.427}
SPL {X  -162.820, Y  +618.758, Z    +0.000, E1   +22.239, E3 +546925.578}
SPL {X  -162.820, Y  +616.062, Z    +0.000, E1   +22.275, E3 +546938.999}
SPL {X  -162.820, Y  +613.536, Z    +0.000, E1   +22.242, E3 +546952.120}
SPL {X  -162.820, Y  +610.461, Z    +0.000, E1   +22.264, E3 +546967.751}
SPL {X  -162.820, Y  +607.796, Z    +0.000, E1   +22.261, E3 +546981.123}
SPL {X  -162.820, Y  +605.178, Z    +0.000, E1   +22.267, E3 +546994.606}
SPL {X  -162.820, Y  +602.350, Z    +0.000, E1   +22.224, E3 +547009.224}
SPL {X  -162.820, Y  +599.842, Z    +0.000, E1   +22.298, E3 +547021.375}
SPL {X  -162.820, Y  +597.194, Z    +0.000, E1   +22.253, E3 +547035.296}
SPL {X  -162.820, Y  +594.115, Z    +0.000, E1   +22.273, E3 +547050.825}
SPL {X  -162.820, Y  +591.721, Z    +0.000, E1   +22.239, E3 +547063.140}
SPL {X  -162.820, Y  +589.492, Z    +0.000, E1   +22.304, E3 +547074.001}
SPL {X  -162.820, Y  +587.447, Z    +0.000, E1   +22.279, E3 +547084.530}
SPL {X  -162.820, Y  +585.192, Z    +0.000, E1   +22.298, E3 +547095.940}
SPL {X  -162.820, Y  +582.610, Z    +0.000, E1   +22.234, E3 +547109.563}
SPL {X  -162.820, Y  +580.317, Z    +0.000, E1   +22.300, E3 +547120.617}
SPL {X  -162.820, Y  +578.878, Z    +0.000, E1   +22.272, E3 +547128.127}
SPL {X  -162.820, Y  +576.856, Z    +0.000, E1   +22.233, E3 +547138.885}
SPL {X  -162.820, Y  +574.811, Z    +0.000, E1   +22.236, E3 +547149.149}
SPL {X  -162.820, Y  +572.645, Z    +0.000, E1   +22.246, E3 +547160.244}
SPL {X  -162.820, Y  +569.475, Z    +0.000, E1   +22.269, E3 +547176.250}
SPL {X  -162.820, Y  +565.838, Z    +0.000, E1   +22.271, E3 +547194.845}
SPL {X  -162.820, Y  +562.162, Z    +0.000, E1   +22.252, E3 +547213.662}
SPL {X  -162.820, Y  +559.515, Z    +0.000, E1   +22.273, E3 +547226.781}
SPL {X  -162.820, Y  +556.723, Z    +0.000, E1   +22.309, E3 +547240.865}
SPL {X  -162.820, Y  +553.294, Z    +0.000, E1   +22.266, E3 +547258.653}
SPL {X  -162.820, Y  +550.136, Z    +0.000, E1   +22.258, E3 +547274.766}
SPL {X  -162.820, Y  +546.694, Z    +0.000, E1   +22.290, E3 +547292.088}
SPL {X  -162.820, Y  +543.558, Z    +0.000, E1   +22.285, E3 +547307.951}
SPL {X  -162.820, Y  +541.633, Z    +0.000, E1   +22.257, E3 +547317.879}
SPL {X  -162.820, Y  +539.116, Z    +0.000, E1   +22.302, E3 +547330.490}
SPL {X  -162.820, Y  +536.913, Z    +0.000, E1   +22.192, E3 +547342.414}
SPL {X  -162.820, Y  +534.880, Z    +0.000, E1   +22.252, E3 +547352.368}
SPL {X  -162.820, Y  +532.896, Z    +0.000, E1   +22.234, E3 +547362.528}
SPL {X  -162.820, Y  +531.056, Z    +0.000, E1   +22.251, E3 +547371.810}
SPL {X  -162.820, Y  +528.708, Z    +0.000, E1   +22.319, E3 +547383.191}
SPL {X  -162.820, Y  +525.932, Z    +0.000, E1   +22.258, E3 +547397.948}
SPL {X  -162.820, Y  +522.524, Z    +0.000, E1   +22.326, E3 +547414.672}
SPL {X  -162.820, Y  +519.457, Z    +0.000, E1   +22.481, E3 +547428.801}
SPL {X  -162.820, Y  +506.285, Z    +0.000, E1   +28.538, E3 +547440.258}
SPL {X  -162.820, Y  +504.441, Z    +0.000, E1   +27.574, E3 +547454.601}
SPL {X  -162.820, Y  +503.215, Z    +0.000, E1   +26.369, E3 +547468.108}
SPL {X  -162.820, Y  +502.265, Z    +0.000, E1   +25.287, E3 +547480.590}
SPL {X  -162.820, Y  +501.060, Z    +0.000, E1   +24.081, E3 +547495.330}
SPL {X  -162.820, Y  +500.336, Z    +0.000, E1   +23.110, E3 +547506.470}
SPL {X  -162.820, Y  +499.240, Z    +0.000, E1   +22.316, E3 +547518.781}
SPL {X  -162.820, Y  +498.027, Z    +0.000, E1   +21.516, E3 +547531.689}
SPL {X  -162.820, Y  +495.897, Z    +0.000, E1   +21.662, E3 +547541.609}
SPL {X  -162.820, Y  +493.717, Z    +0.000, E1   +21.704, E3 +547552.715}
SPL {X  -162.820, Y  +491.396, Z    +0.000, E1   +21.707, E3 +547564.839}
SPL {X  -162.820, Y  +488.560, Z    +0.000, E1   +21.695, E3 +547579.949}
SPL {X  -162.820, Y  +485.661, Z    +0.000, E1   +21.712, E3 +547594.834}
SPL {X  -162.820, Y  +483.668, Z    +0.000, E1   +21.664, E3 +547605.661}
SPL {X  -162.820, Y  +481.739, Z    +0.000, E1   +21.704, E3 +547615.375}
SPL {X  -162.820, Y  +479.894, Z    +0.000, E1   +21.695, E3 +547625.162}
SPL {X  -162.820, Y  +477.685, Z    +0.000, E1   +21.656, E3 +547637.100}
SPL {X  -162.820, Y  +475.419, Z    +0.000, E1   +21.711, E3 +547648.453}
SPL {X  -162.820, Y  +473.301, Z    +0.000, E1   +21.712, E3 +547659.550}
SPL {X  -162.820, Y  +470.965, Z    +0.000, E1   +21.700, E3 +547671.895}
SPL {X  -162.820, Y  +469.036, Z    +0.000, E1   +21.695, E3 +547681.938}
SPL {X  -162.820, Y  +467.138, Z    +0.000, E1   +21.678, E3 +547692.110}
SPL {X  -162.820, Y  +465.011, Z    +0.000, E1   +21.692, E3 +547703.093}
SPL {X  -162.820, Y  +462.669, Z    +0.000, E1   +21.752, E3 +547714.873}
SPL {X  -162.820, Y  +460.725, Z    +0.000, E1   +21.689, E3 +547725.486}
SPL {X  -162.820, Y  +458.666, Z    +0.000, E1   +21.695, E3 +547736.298}
SPL {X  -162.820, Y  +456.431, Z    +0.000, E1   +21.708, E3 +547747.827}
SPL {X  -162.820, Y  +453.609, Z    +0.000, E1   +21.757, E3 +547762.361}
SPL {X  -162.820, Y  +450.610, Z    +0.000, E1   +21.698, E3 +547778.418}
SPL {X  -162.820, Y  +448.170, Z    +0.000, E1   +21.667, E3 +547791.439}
SPL {X  -162.820, Y  +445.508, Z    +0.000, E1   +21.732, E3 +547804.957}
SPL {X  -162.820, Y  +442.443, Z    +0.000, E1   +21.712, E3 +547821.078}
SPL {X  -162.820, Y  +439.933, Z    +0.000, E1   +21.690, E3 +547834.358}
SPL {X  -162.820, Y  +437.628, Z    +0.000, E1   +21.678, E3 +547846.546}
SPL {X  -162.820, Y  +434.473, Z    +0.000, E1   +21.747, E3 +547862.643}
SPL {X  -162.820, Y  +431.492, Z    +0.000, E1   +21.686, E3 +547878.591}
SPL {X  -162.820, Y  +429.074, Z    +0.000, E1   +21.710, E3 +547891.043}
SPL {X  -162.820, Y  +426.023, Z    +0.000, E1   +21.718, E3 +547907.111}
SPL {X  -162.820, Y  +422.986, Z    +0.000, E1   +21.685, E3 +547923.159}
SPL {X  -162.820, Y  +420.528, Z    +0.000, E1   +21.706, E3 +547935.809}
SPL {X  -162.820, Y  +418.116, Z    +0.000, E1   +21.761, E3 +547947.956}
SPL {X  -162.820, Y  +416.127, Z    +0.000, E1   +21.715, E3 +547958.661}
SPL {X  -162.820, Y  +414.361, Z    +0.000, E1   +21.613, E3 +547968.848}
SPL {X  -162.820, Y  +411.450, Z    +0.000, E1   +21.710, E3 +547983.422}
SPL {X  -162.820, Y  +408.590, Z    +0.000, E1   +21.735, E3 +547998.047}
SPL {X  -162.820, Y  +406.238, Z    +0.000, E1   +21.697, E3 +548010.696}
SPL {X  -162.820, Y  +403.166, Z    +0.000, E1   +21.746, E3 +548026.502}
SPL {X  -162.820, Y  +400.348, Z    +0.000, E1   +21.713, E3 +548041.337}
SPL {X  -162.820, Y  +398.298, Z    +0.000, E1   +21.721, E3 +548051.953}
SPL {X  -162.820, Y  +396.371, Z    +0.000, E1   +21.713, E3 +548062.134}
SPL {X  -162.820, Y  +394.508, Z    +0.000, E1   +21.616, E3 +548072.690}
SPL {X  -162.820, Y  +391.777, Z    +0.000, E1   +21.714, E3 +548086.349}
SPL {X  -162.820, Y  +388.822, Z    +0.000, E1   +21.717, E3 +548101.669}
SPL {X  -162.820, Y  +386.818, Z    +0.000, E1   +21.679, E3 +548112.409}
SPL {X  -162.820, Y  +384.697, Z    +0.000, E1   +21.693, E3 +548123.479}
SPL {X  -162.820, Y  +382.288, Z    +0.000, E1   +21.742, E3 +548135.603}
SPL {X  -162.817, Y  +379.520, Z    +0.000, E1   +21.723, E3 +548150.440}
SPL {X  -162.776, Y  +376.710, Z    +0.000, E1   +21.698, E3 +548165.179}
SPL {X  -162.707, Y  +374.438, Z    +0.000, E1   +21.688, E3 +548177.183}
SPL {X  -162.607, Y  +372.171, Z    +0.000, E1   +21.692, E3 +548188.983}
SPL {X  -162.494, Y  +370.197, Z    +0.000, E1   +21.655, E3 +548199.609}
SPL {X  -162.349, Y  +368.131, Z    +0.000, E1   +21.624, E3 +548210.727}
SPL {X  -162.161, Y  +365.866, Z    +0.000, E1   +21.642, E3 +548222.412}
SPL {X  -161.927, Y  +363.466, Z    +0.000, E1   +21.730, E3 +548234.184}
SPL {X  -160.290, Y  +351.907, Z    +0.000, E1   +27.562, E3 +548241.761}
SPL {X  -160.281, Y  +351.857, Z    +0.000, E1   +24.243, E3 +548271.175}
ENDSPLINE

SPLINE
SPL {X  -161.833, Y  +362.603, Z    +0.000, E1   +17.021, E3 +548285.870}
ENDSPLINE

SPLINE
SPL {X  -160.786, Y  +354.842, Z    +0.000, E1   +19.274, E3 +548318.026}
ENDSPLINE

SPLINE
SPL {X  -162.485, Y  +370.062, Z    +0.000, E1   +10.606, E3 +548324.404}
SPL {X  -162.820, Y  +381.311, Z    +0.000, E1    +4.054, E3 +548314.759}
SPL {X  -162.820, Y  +390.142, Z    +0.000, E1    -2.185, E3 +548315.087}
SPL {X  -162.820, Y  +393.415, Z    +0.000, E1    -4.587, E3 +548320.195}
SPL {X  -162.820, Y  +399.630, Z    +0.000, E1    -9.426, E3 +548322.124}
SPL {X  -162.820, Y  +408.127, Z    +0.000, E1   -18.417, E3 +548308.413}
SPL {X  -162.820, Y  +420.083, Z    +0.000, E1   -24.325, E3 +548328.888}
SPL {X  -162.820, Y  +428.527, Z    +0.000, E1   -26.988, E3 +548346.180}
SPL {X  -162.820, Y  +431.336, Z    +0.000, E1   -24.162, E3 +548376.390}
SPL {X  -162.820, Y  +432.048, Z    +0.000, E1   -22.832, E3 +548390.894}
SPL {X  -162.820, Y  +434.888, Z    +0.000, E1   -22.823, E3 +548404.844}
SPL {X  -162.820, Y  +436.834, Z    +0.000, E1   -22.779, E3 +548414.804}
SPL {X  -162.820, Y  +438.868, Z    +0.000, E1   -22.837, E3 +548424.457}
SPL {X  -162.820, Y  +441.351, Z    +0.000, E1   -22.805, E3 +548437.033}
SPL {X  -162.820, Y  +443.809, Z    +0.000, E1   -22.804, E3 +548449.199}
SPL {X  -162.820, Y  +447.077, Z    +0.000, E1   -22.869, E3 +548465.009}
SPL {X  -162.820, Y  +449.911, Z    +0.000, E1   -22.774, E3 +548479.619}
SPL {X  -162.820, Y  +451.861, Z    +0.000, E1   -22.750, E3 +548489.466}
SPL {X  -162.820, Y  +454.167, Z    +0.000, E1   -22.842, E3 +548500.196}
SPL {X  -162.820, Y  +456.529, Z    +0.000, E1   -22.855, E3 +548511.724}
SPL {X  -162.820, Y  +458.725, Z    +0.000, E1   -22.793, E3 +548523.129}
SPL {X  -162.820, Y  +461.700, Z    +0.000, E1   -22.822, E3 +548537.751}
SPL {X  -162.820, Y  +464.633, Z    +0.000, E1   -22.813, E3 +548552.248}
SPL {X  -162.820, Y  +466.699, Z    +0.000, E1   -22.824, E3 +548562.294}
SPL {X  -162.820, Y  +468.655, Z    +0.000, E1   -22.858, E3 +548571.738}
SPL {X  -162.820, Y  +470.892, Z    +0.000, E1   -22.837, E3 +548582.976}
SPL {X  -162.820, Y  +473.485, Z    +0.000, E1   -22.806, E3 +548596.175}
SPL {X  -162.820, Y  +475.738, Z    +0.000, E1   -22.728, E3 +548607.840}
SPL {X  -162.820, Y  +478.177, Z    +0.000, E1   -22.834, E3 +548619.179}
SPL {X  -162.820, Y  +481.034, Z    +0.000, E1   -22.831, E3 +548633.317}
SPL {X  -162.820, Y  +483.391, Z    +0.000, E1   -22.793, E3 +548645.253}
SPL {X  -162.820, Y  +486.307, Z    +0.000, E1   -22.833, E3 +548659.507}
SPL {X  -162.820, Y  +489.750, Z    +0.000, E1   -22.832, E3 +548676.577}
SPL {X  -162.820, Y  +492.546, Z    +0.000, E1   -22.823, E3 +548690.335}
SPL {X  -162.820, Y  +495.526, Z    +0.000, E1   -22.833, E3 +548705.218}
SPL {X  -162.820, Y  +499.330, Z    +0.000, E1   -22.841, E3 +548723.999}
SPL {X  -162.820, Y  +503.049, Z    +0.000, E1   -22.823, E3 +548742.548}
SPL {X  -162.820, Y  +506.908, Z    +0.000, E1   -22.877, E3 +548761.218}
SPL {X  -162.820, Y  +510.068, Z    +0.000, E1   -22.761, E3 +548777.690}
SPL {X  -162.820, Y  +512.359, Z    +0.000, E1   -22.823, E3 +548788.421}
SPL {X  -162.820, Y  +513.873, Z    +0.000, E1   -22.800, E3 +548796.108}
SPL {X  -162.820, Y  +516.100, Z    +0.000, E1   -22.809, E3 +548807.184}
SPL {X  -162.820, Y  +518.662, Z    +0.000, E1   -22.847, E3 +548819.483}
SPL {X  -162.820, Y  +520.641, Z    +0.000, E1   -22.790, E3 +548829.724}
SPL {X  -162.820, Y  +523.535, Z    +0.000, E1   -22.857, E3 +548843.693}
SPL {X  -162.820, Y  +526.661, Z    +0.000, E1   -22.801, E3 +548859.517}
SPL {X  -162.820, Y  +528.725, Z    +0.000, E1   -22.770, E3 +548869.886}
SPL {X  -162.820, Y  +530.303, Z    +0.000, E1   -22.798, E3 +548877.505}
SPL {X  -162.820, Y  +532.614, Z    +0.000, E1   -22.828, E3 +548888.774}
SPL {X  -162.820, Y  +534.838, Z    +0.000, E1   -22.864, E3 +548899.403}
SPL {X  -162.820, Y  +536.882, Z    +0.000, E1   -22.782, E3 +548910.258}
SPL {X  -162.820, Y  +539.194, Z    +0.000, E1   -22.826, E3 +548921.306}
SPL {X  -162.820, Y  +541.555, Z    +0.000, E1   -22.817, E3 +548933.120}
SPL {X  -162.820, Y  +543.728, Z    +0.000, E1   -22.799, E3 +548943.978}
SPL {X  -162.820, Y  +545.925, Z    +0.000, E1   -22.803, E3 +548954.848}
SPL {X  -162.820, Y  +549.071, Z    +0.000, E1   -22.836, E3 +548970.375}
SPL {X  -162.820, Y  +553.089, Z    +0.000, E1   -22.838, E3 +548990.275}
SPL {X  -162.820, Y  +556.430, Z    +0.000, E1   -22.821, E3 +549006.776}
SPL {X  -162.820, Y  +559.675, Z    +0.000, E1   -22.837, E3 +549022.857}
SPL {X  -162.820, Y  +562.799, Z    +0.000, E1   -22.814, E3 +549038.363}
SPL {X  -162.820, Y  +565.170, Z    +0.000, E1   -22.801, E3 +549050.188}
SPL {X  -162.820, Y  +568.020, Z    +0.000, E1   -22.787, E3 +549064.574}
SPL {X  -162.820, Y  +570.992, Z    +0.000, E1   -22.834, E3 +549078.794}
SPL {X  -162.820, Y  +572.901, Z    +0.000, E1   -22.775, E3 +549088.662}
SPL {X  -162.820, Y  +575.638, Z    +0.000, E1   -22.855, E3 +549101.771}
SPL {X  -162.820, Y  +578.553, Z    +0.000, E1   -22.801, E3 +549116.484}
SPL {X  -162.820, Y  +581.064, Z    +0.000, E1   -22.823, E3 +549128.768}
SPL {X  -162.820, Y  +583.435, Z    +0.000, E1   -22.808, E3 +549140.590}
SPL {X  -162.820, Y  +585.410, Z    +0.000, E1   -22.764, E3 +549150.726}
SPL {X  -162.820, Y  +587.676, Z    +0.000, E1   -22.853, E3 +549161.240}
SPL {X  -162.820, Y  +589.682, Z    +0.000, E1   -22.776, E3 +549171.770}
SPL {X  -162.820, Y  +591.720, Z    +0.000, E1   -22.868, E3 +549181.081}
SPL {X  -162.820, Y  +593.650, Z    +0.000, E1   -22.810, E3 +549191.151}
SPL {X  -162.820, Y  +595.830, Z    +0.000, E1   -22.828, E3 +549201.767}
SPL {X  -162.820, Y  +598.094, Z    +0.000, E1   -22.843, E3 +549212.880}
SPL {X  -162.820, Y  +600.420, Z    +0.000, E1   -22.826, E3 +549224.511}
SPL {X  -162.820, Y  +602.573, Z    +0.000, E1   -22.830, E3 +549235.096}
SPL {X  -162.820, Y  +604.828, Z    +0.000, E1   -22.784, E3 +549246.734}
SPL {X  -162.820, Y  +608.133, Z    +0.000, E1   -22.831, E3 +549262.852}
SPL {X  -162.820, Y  +611.103, Z    +0.000, E1   -22.785, E3 +549277.778}
SPL {X  -162.820, Y  +613.294, Z    +0.000, E1   -22.780, E3 +549288.651}
SPL {X  -162.820, Y  +615.356, Z    +0.000, E1   -22.799, E3 +549298.708}
SPL {X  -162.820, Y  +617.439, Z    +0.000, E1   -22.808, E3 +549308.966}
SPL {X  -162.820, Y  +619.665, Z    +0.000, E1   -22.817, E3 +549319.934}
SPL {X  -162.820, Y  +621.733, Z    +0.000, E1   -22.759, E3 +549330.659}
SPL {X  -162.820, Y  +624.076, Z    +0.000, E1   -22.774, E3 +549342.164}
SPL {X  -162.820, Y  +627.244, Z    +0.000, E1   -22.803, E3 +549357.846}
SPL {X  -162.820, Y  +630.349, Z    +0.000, E1   -22.766, E3 +549373.378}
SPL {X  -162.820, Y  +632.572, Z    +0.000, E1   -22.785, E3 +549384.185}
SPL {X  -162.820, Y  +634.507, Z    +0.000, E1   -22.784, E3 +549393.823}
SPL {X  -162.820, Y  +636.863, Z    +0.000, E1   -22.760, E3 +549405.746}
SPL {X  -162.820, Y  +640.111, Z    +0.000, E1   -22.809, E3 +549421.628}
SPL {X  -162.820, Y  +643.449, Z    +0.000, E1   -22.796, E3 +549438.146}
SPL {X  -162.820, Y  +645.630, Z    +0.000, E1   -22.795, E3 +549448.842}
SPL {X  -162.820, Y  +647.561, Z    +0.000, E1   -22.705, E3 +549459.293}
SPL {X  -162.820, Y  +649.758, Z    +0.000, E1   -22.780, E3 +549469.483}
SPL {X  -162.820, Y  +651.708, Z    +0.000, E1   -22.810, E3 +549478.977}
SPL {X  -162.820, Y  +653.898, Z    +0.000, E1   -22.796, E3 +549489.898}
SPL {X  -162.820, Y  +656.161, Z    +0.000, E1   -22.812, E3 +549501.020}
SPL {X  -162.820, Y  +658.384, Z    +0.000, E1   -22.822, E3 +549511.886}
SPL {X  -162.820, Y  +660.215, Z    +0.000, E1   -22.649, E3 +549522.477}
SPL {X  -162.820, Y  +662.823, Z    +0.000, E1   -22.799, E3 +549534.184}
SPL {X  -162.820, Y  +665.112, Z    +0.000, E1   -22.835, E3 +549545.239}
SPL {X  -162.820, Y  +667.016, Z    +0.000, E1   -22.823, E3 +549554.667}
SPL {X  -162.820, Y  +668.960, Z    +0.000, E1   -22.773, E3 +549564.835}
SPL {X  -162.820, Y  +672.333, Z    +0.000, E1   -22.837, E3 +549581.171}
SPL {X  -162.812, Y  +675.071, Z    +0.000, E1   -22.742, E3 +549595.316}
SPL {X  -162.773, Y  +677.428, Z    +0.000, E1   -22.762, E3 +549606.913}
SPL {X  -162.691, Y  +679.987, Z    +0.000, E1   -22.794, E3 +549619.327}
SPL {X  -162.604, Y  +681.880, Z    +0.000, E1   -22.691, E3 +549629.487}
SPL {X  -162.458, Y  +684.346, Z    +0.000, E1   -22.764, E3 +549641.281}
SPL {X  -162.296, Y  +686.547, Z    +0.000, E1   -22.660, E3 +549652.898}
SPL {X  -162.090, Y  +688.902, Z    +0.000, E1   -22.700, E3 +549664.406}
SPL {X  -161.474, Y  +694.390, Z    +0.000, E1   -24.298, E3 +549677.761}
SPL {X  -158.730, Y  +709.763, Z    +0.000, E1   -31.225, E3 +549689.100}
ENDSPLINE

SPLINE
SPL {X  -160.932, Y  +698.225, Z    +0.000, E1   -21.712, E3 +549720.209}
SPL {X  -161.691, Y  +692.643, Z    +0.000, E1   -17.369, E3 +549737.092}
SPL {X  -162.534, Y  +683.153, Z    +0.000, E1   -10.475, E3 +549762.559}
SPL {X  -162.820, Y  +667.630, Z    +0.000, E1    -0.882, E3 +549756.535}
SPL {X  -162.820, Y  +661.883, Z    +0.000, E1    +3.373, E3 +549761.979}
SPL {X  -162.820, Y  +653.808, Z    +0.000, E1    +9.891, E3 +549759.670}
SPL {X  -162.820, Y  +632.548, Z    +0.000, E1   +27.446, E3 +549756.207}
ENDSPLINE

SPLINE
SPL {X  -162.820, Y  +638.080, Z    +0.000, E1   +18.858, E3 +549783.955}
ENDSPLINE

SPLINE
SPL {X  -162.820, Y  +623.278, Z    +0.000, E1   +28.723, E3 +549785.526}
SPL {X  -162.820, Y  +618.658, Z    +0.000, E1   +26.841, E3 +549814.135}
ENDSPLINE

SPLINE
SPL {X  -162.820, Y  +623.685, Z    +0.000, E1   +22.346, E3 +549826.441}
ENDSPLINE

